LIN {X 0,Y 552.983,Z 1250.338,A -85,B 0,C 180,E1 26531.445,E2 26531.445} C_VEL
LIN {X 0,Y 553.442,Z 1236.475,A -85,B 0,C 180,E1 26529.594,E2 26529.594} C_VEL
LIN {X 0,Y 554.004,Z 1220.765,A -85,B 0,C 180,E1 26527.797,E2 26527.797} C_VEL
LIN {X 0,Y 554.663,Z 1203.891,A -85,B 0,C 180,E1 26526.129,E2 26526.129} C_VEL
LIN {X 0,Y 555.379,Z 1185.775,A -85,B 0,C 180,E1 26524.588,E2 26524.588} C_VEL
LIN {X 0,Y 556.106,Z 1167.101,A -85,B 0,C 180,E1 26523.232,E2 26523.232} C_VEL
LIN {X 0,Y 556.817,Z 1147.774,A -85,B 0,C 180,E1 26522.053,E2 26522.053} C_VEL
LIN {X 0,Y 557.493,Z 1127.887,A -85,B 0,C 180,E1 26521.038,E2 26521.038} C_VEL
LIN {X 0,Y 558.107,Z 1108.035,A -85,B 0,C 180,E1 26520.219,E2 26520.219} C_VEL
LIN {X 0,Y 558.611,Z 1086.262,A -85,B 0,C 180,E1 26519.523,E2 26519.523} C_VEL
LIN {X 0,Y 559.061,Z 1064.401,A -85,B 0,C 180,E1 26519.023,E2 26519.023} C_VEL
LIN {X 0,Y 560.686,Z 838.01,A -85,B 0,C 180,E1 26515.721,E2 26515.721} C_VEL
LIN {X 0,Y 561.006,Z 768.004,A -85,B 0,C 180,E1 26514.675,E2 26514.675} C_VEL
LIN {X 0,Y 559.471,Z 758.813,A -85,B 0,C 180,E1 26514.405,E2 26514.405} C_VEL
LIN {X 0,Y 560.826,Z 708.184,A -85,B 0,C 180,E1 26511.131,E2 26511.131} C_VEL
LIN {X 0,Y 561.473,Z 685.988,A -85,B 0,C 180,E1 26509.656,E2 26509.656} C_VEL
LIN {X 0,Y 552.413,Z 666.42,A -85,B 0,C 180,E1 26507.601,E2 26507.601} C_VEL
LIN {X 0,Y 552.326,Z 665.917,A -85,B 0,C 180,E1 26507.248,E2 26507.248} C_VEL
LIN {X 0,Y 552.322,Z 665.911,A -85,B 0,C 180,E1 26504.039,E2 26504.039} C_VEL
LIN {X 0,Y 552.331,Z 665.93,A -85,B 0,C 180,E1 26500.669,E2 26500.669} C_VEL
LIN {X 0,Y 552.333,Z 665.926,A -85,B 0,C 180,E1 26497.332,E2 26497.332} C_VEL
LIN {X 0,Y 552.336,Z 665.92,A -85,B 0,C 180,E1 26493.812,E2 26493.812} C_VEL
LIN {X 0,Y 552.328,Z 665.927,A -85,B 0,C 180,E1 26490.456,E2 26490.456} C_VEL
LIN {X 0,Y 552.327,Z 665.93,A -85,B 0,C 180,E1 26487.141,E2 26487.141} C_VEL
LIN {X 0,Y 552.324,Z 665.931,A -85,B 0,C 180,E1 26483.809,E2 26483.809} C_VEL
LIN {X 0,Y 552.324,Z 665.931,A -85,B 0,C 180,E1 26480.56,E2 26480.56} C_VEL
LIN {X 0,Y 552.323,Z 665.931,A -85,B 0,C 180,E1 26477.27,E2 26477.27} C_VEL
LIN {X 0,Y 552.324,Z 665.932,A -85,B 0,C 180,E1 26474.004,E2 26474.004} C_VEL
LIN {X 0,Y 552.324,Z 665.93,A -85,B 0,C 180,E1 26470.746,E2 26470.746} C_VEL
LIN {X 0,Y 552.327,Z 665.932,A -85,B 0,C 180,E1 26467.489,E2 26467.489} C_VEL
LIN {X 0,Y 552.325,Z 665.928,A -85,B 0,C 180,E1 26464.152,E2 26464.152} C_VEL
LIN {X 0,Y 552.345,Z 665.934,A -85,B 0,C 180,E1 26460.726,E2 26460.726} C_VEL
LIN {X 0,Y 552.337,Z 665.924,A -85,B 0,C 180,E1 26457.302,E2 26457.302} C_VEL
LIN {X 0,Y 552.332,Z 665.924,A -85,B 0,C 180,E1 26453.869,E2 26453.869} C_VEL
LIN {X 0,Y 552.335,Z 665.935,A -85,B 0,C 180,E1 26450.518,E2 26450.518} C_VEL
LIN {X 0,Y 552.324,Z 665.928,A -85,B 0,C 180,E1 26447.134,E2 26447.134} C_VEL
LIN {X 0,Y 552.341,Z 665.931,A -85,B 0,C 180,E1 26443.813,E2 26443.813} C_VEL
LIN {X 0,Y 552.326,Z 665.928,A -85,B 0,C 180,E1 26440.433,E2 26440.433} C_VEL
LIN {X 0,Y 552.338,Z 665.929,A -85,B 0,C 180,E1 26437.095,E2 26437.095} C_VEL
LIN {X 0,Y 552.336,Z 665.932,A -85,B 0,C 180,E1 26433.672,E2 26433.672} C_VEL
LIN {X 0,Y 552.339,Z 665.926,A -85,B 0,C 180,E1 26432.662,E2 26432.662} C_VEL
LIN {X 0,Y 551.37,Z 666.049,A -85,B 0,C 180,E1 26431.863,E2 26431.863} C_VEL
LIN {X 0,Y 544.853,Z 666.84,A -85,B 0,C 180,E1 26429.562,E2 26429.562} C_VEL
LIN {X 0,Y 544.401,Z 666.902,A -85,B 0,C 180,E1 26429.035,E2 26429.035} C_VEL
LIN {X 0,Y 544.387,Z 666.919,A -85,B 0,C 180,E1 26425.677,E2 26425.677} C_VEL
LIN {X 0,Y 544.387,Z 666.91,A -85,B 0,C 180,E1 26422.294,E2 26422.294} C_VEL
LIN {X 0,Y 544.386,Z 666.922,A -85,B 0,C 180,E1 26419.012,E2 26419.012} C_VEL
LIN {X 0,Y 544.387,Z 666.922,A -85,B 0,C 180,E1 26415.738,E2 26415.738} C_VEL
LIN {X 0,Y 544.393,Z 666.905,A -85,B 0,C 180,E1 26412.379,E2 26412.379} C_VEL
LIN {X 0,Y 544.391,Z 666.91,A -85,B 0,C 180,E1 26409.022,E2 26409.022} C_VEL
LIN {X 0,Y 544.427,Z 667.108,A -85,B 0,C 180,E1 26405.862,E2 26405.862} C_VEL
LIN {X 0,Y 544.787,Z 668.547,A -85,B 0,C 180,E1 26405.695,E2 26405.695} C_VEL
LIN {X 0,Y 554.114,Z 684.335,A -85,B 0,C 180,E1 26404.755,E2 26404.755} C_VEL
LIN {X 0,Y 552.272,Z 907.322,A -85,B 0,C 180,E1 26401.482,E2 26401.482} C_VEL
LIN {X 0,Y 551.925,Z 928.962,A -85,B 0,C 180,E1 26401.05,E2 26401.05} C_VEL
LIN {X 0,Y 551.302,Z 950.414,A -85,B 0,C 180,E1 26400.423,E2 26400.423} C_VEL
LIN {X 0,Y 550.639,Z 971.812,A -85,B 0,C 180,E1 26399.596,E2 26399.596} C_VEL
LIN {X 0,Y 549.869,Z 991.939,A -85,B 0,C 180,E1 26398.628,E2 26398.628} C_VEL
LIN {X 0,Y 549.069,Z 1011.113,A -85,B 0,C 180,E1 26397.497,E2 26397.497} C_VEL
LIN {X 0,Y 548.16,Z 1031.38,A -85,B 0,C 180,E1 26396.077,E2 26396.077} C_VEL
LIN {X 0,Y 547.353,Z 1049.163,A -85,B 0,C 180,E1 26394.612,E2 26394.612} C_VEL
LIN {X 0,Y 546.577,Z 1066.575,A -85,B 0,C 180,E1 26392.932,E2 26392.932} C_VEL
LIN {X 0,Y 545.879,Z 1082.44,A -85,B 0,C 180,E1 26391.151,E2 26391.151} C_VEL
LIN {X 0,Y 545.271,Z 1097.705,A -85,B 0,C 180,E1 26389.161,E2 26389.161} C_VEL
LIN {X 0,Y 544.81,Z 1110.729,A -85,B 0,C 180,E1 26387.185,E2 26387.185} C_VEL
LIN {X 0,Y 544.454,Z 1122.312,A -85,B 0,C 180,E1 26385.116,E2 26385.116} C_VEL
LIN {X 0,Y 544.213,Z 1132.49,A -85,B 0,C 180,E1 26382.952,E2 26382.952} C_VEL
LIN {X 0,Y 544.065,Z 1140.901,A -85,B 0,C 180,E1 26380.804,E2 26380.804} C_VEL
LIN {X 0,Y 543.977,Z 1147.547,A -85,B 0,C 180,E1 26378.668,E2 26378.668} C_VEL
LIN {X 0,Y 543.925,Z 1153.108,A -85,B 0,C 180,E1 26376.332,E2 26376.332} C_VEL
LIN {X 0,Y 543.908,Z 1156.822,A -85,B 0,C 180,E1 26374.111,E2 26374.111} C_VEL
LIN {X 0,Y 543.901,Z 1158.854,A -85,B 0,C 180,E1 26371.896,E2 26371.896} C_VEL
LIN {X 0,Y 543.898,Z 1159.427,A -85,B 0,C 180,E1 26369.579,E2 26369.579} C_VEL
LIN {X 0,Y 543.898,Z 1158.439,A -85,B 0,C 180,E1 26367.366,E2 26367.366} C_VEL
LIN {X 0,Y 543.904,Z 1155.79,A -85,B 0,C 180,E1 26365.11,E2 26365.11} C_VEL
LIN {X 0,Y 543.929,Z 1151.778,A -85,B 0,C 180,E1 26362.926,E2 26362.926} C_VEL
LIN {X 0,Y 543.988,Z 1146.167,A -85,B 0,C 180,E1 26360.757,E2 26360.757} C_VEL
LIN {X 0,Y 544.096,Z 1138.463,A -85,B 0,C 180,E1 26358.446,E2 26358.446} C_VEL
LIN {X 0,Y 544.28,Z 1129.612,A -85,B 0,C 180,E1 26356.292,E2 26356.292} C_VEL
LIN {X 0,Y 544.552,Z 1119.051,A -85,B 0,C 180,E1 26354.18,E2 26354.18} C_VEL
LIN {X 0,Y 544.961,Z 1106.455,A -85,B 0,C 180,E1 26352.048,E2 26352.048} C_VEL
LIN {X 0,Y 545.461,Z 1092.757,A -85,B 0,C 180,E1 26350.066,E2 26350.066} C_VEL
LIN {X 0,Y 546.099,Z 1077.486,A -85,B 0,C 180,E1 26348.167,E2 26348.167} C_VEL
LIN {X 0,Y 546.814,Z 1060.807,A -85,B 0,C 180,E1 26346.395,E2 26346.395} C_VEL
LIN {X 0,Y 547.631,Z 1042.986,A -85,B 0,C 180,E1 26344.766,E2 26344.766} C_VEL
LIN {X 0,Y 548.53,Z 1023.392,A -85,B 0,C 180,E1 26343.242,E2 26343.242} C_VEL
LIN {X 0,Y 549.377,Z 1004.059,A -85,B 0,C 180,E1 26341.969,E2 26341.969} C_VEL
LIN {X 0,Y 550.159,Z 984.662,A -85,B 0,C 180,E1 26340.913,E2 26340.913} C_VEL
LIN {X 0,Y 550.925,Z 962.845,A -85,B 0,C 180,E1 26339.941,E2 26339.941} C_VEL
LIN {X 0,Y 551.604,Z 941.595,A -85,B 0,C 180,E1 26339.203,E2 26339.203} C_VEL
LIN {X 0,Y 552.071,Z 920.027,A -85,B 0,C 180,E1 26338.66,E2 26338.66} C_VEL
LIN {X 0,Y 552.445,Z 890.261,A -85,B 0,C 180,E1 26338.174,E2 26338.174} C_VEL
LIN {X 0,Y 554.083,Z 683.904,A -85,B 0,C 180,E1 26335.146,E2 26335.146} C_VEL
LIN {X 0,Y 545.839,Z 670.561,A -85,B 0,C 180,E1 26334.331,E2 26334.331} C_VEL
LIN {X 0,Y 544.5,Z 667.51,A -85,B 0,C 180,E1 26334.127,E2 26334.127} C_VEL
LIN {X 0,Y 544.399,Z 666.917,A -85,B 0,C 180,E1 26333.876,E2 26333.876} C_VEL
LIN {X 0,Y 544.386,Z 666.914,A -85,B 0,C 180,E1 26330.48,E2 26330.48} C_VEL
LIN {X 0,Y 544.396,Z 666.906,A -85,B 0,C 180,E1 26327.123,E2 26327.123} C_VEL
LIN {X 0,Y 544.4,Z 666.909,A -85,B 0,C 180,E1 26323.676,E2 26323.676} C_VEL
LIN {X 0,Y 544.393,Z 666.919,A -85,B 0,C 180,E1 26320.18,E2 26320.18} C_VEL
LIN {X 0,Y 544.385,Z 666.904,A -85,B 0,C 180,E1 26316.781,E2 26316.781} C_VEL
LIN {X 0,Y 544.389,Z 666.922,A -85,B 0,C 180,E1 26313.436,E2 26313.436} C_VEL
LIN {X 0,Y 544.383,Z 666.898,A -85,B 0,C 180,E1 26310.094,E2 26310.094} C_VEL
LIN {X 0,Y 544.398,Z 666.922,A -85,B 0,C 180,E1 26306.742,E2 26306.742} C_VEL
LIN {X 0,Y 544.401,Z 666.915,A -85,B 0,C 180,E1 26303.258,E2 26303.258} C_VEL
LIN {X 0,Y 544.395,Z 666.919,A -85,B 0,C 180,E1 26299.752,E2 26299.752} C_VEL
LIN {X 0,Y 544.4,Z 666.919,A -85,B 0,C 180,E1 26296.43,E2 26296.43} C_VEL
LIN {X 0,Y 544.386,Z 666.918,A -85,B 0,C 180,E1 26293.057,E2 26293.057} C_VEL
LIN {X 0,Y 544.403,Z 666.922,A -85,B 0,C 180,E1 26289.728,E2 26289.728} C_VEL
LIN {X 0,Y 544.385,Z 666.912,A -85,B 0,C 180,E1 26286.433,E2 26286.433} C_VEL
LIN {X 0,Y 544.393,Z 666.918,A -85,B 0,C 180,E1 26283.053,E2 26283.053} C_VEL
LIN {X 0,Y 544.393,Z 666.919,A -85,B 0,C 180,E1 26279.684,E2 26279.684} C_VEL
LIN {X 0,Y 544.4,Z 666.917,A -85,B 0,C 180,E1 26276.209,E2 26276.209} C_VEL
LIN {X 0,Y 544.406,Z 666.918,A -85,B 0,C 180,E1 26272.72,E2 26272.72} C_VEL
LIN {X 0,Y 544.386,Z 666.918,A -85,B 0,C 180,E1 26269.292,E2 26269.292} C_VEL
LIN {X 0,Y 544.385,Z 666.919,A -85,B 0,C 180,E1 26265.97,E2 26265.97} C_VEL
LIN {X 0,Y 544.385,Z 666.92,A -85,B 0,C 180,E1 26262.69,E2 26262.69} C_VEL
LIN {X 0,Y 544.388,Z 666.919,A -85,B 0,C 180,E1 26259.351,E2 26259.351} C_VEL
LIN {X 0,Y 544.39,Z 666.918,A -85,B 0,C 180,E1 26256.053,E2 26256.053} C_VEL
LIN {X 0,Y 544.397,Z 666.918,A -85,B 0,C 180,E1 26252.667,E2 26252.667} C_VEL
LIN {X 0,Y 544.401,Z 666.922,A -85,B 0,C 180,E1 26249.175,E2 26249.175} C_VEL
LIN {X 0,Y 544.388,Z 666.911,A -85,B 0,C 180,E1 26245.738,E2 26245.738} C_VEL
LIN {X 0,Y 544.386,Z 666.914,A -85,B 0,C 180,E1 26242.427,E2 26242.427} C_VEL
LIN {X 0,Y 544.386,Z 666.911,A -85,B 0,C 180,E1 26239.167,E2 26239.167} C_VEL
LIN {X 0,Y 544.382,Z 666.897,A -85,B 0,C 180,E1 26235.885,E2 26235.885} C_VEL
LIN {X 0,Y 544.429,Z 667.133,A -85,B 0,C 180,E1 26233.02,E2 26233.02} C_VEL
LIN {X 0,Y 545.459,Z 670.023,A -85,B 0,C 180,E1 26232.688,E2 26232.688} C_VEL
LIN {X 0,Y 554.761,Z 689.588,A -85,B 0,C 180,E1 26230.644,E2 26230.644} C_VEL
LIN {X 0,Y 553.444,Z 733.168,A -85,B 0,C 180,E1 26227.765,E2 26227.765} C_VEL
LIN {X 0,Y 552.785,Z 759.73,A -85,B 0,C 180,E1 26226.062,E2 26226.062} C_VEL
LIN {X 0,Y 554.646,Z 771.849,A -85,B 0,C 180,E1 26225.732,E2 26225.732} C_VEL
LIN {X 0,Y 552.714,Z 1006.467,A -85,B 0,C 180,E1 26222.271,E2 26222.271} C_VEL
LIN {X 0,Y 552.174,Z 1066.601,A -85,B 0,C 180,E1 26221.367,E2 26221.367} C_VEL
LIN {X 0,Y 551.644,Z 1088.329,A -85,B 0,C 180,E1 26220.844,E2 26220.844} C_VEL
LIN {X 0,Y 551.02,Z 1110.245,A -85,B 0,C 180,E1 26220.113,E2 26220.113} C_VEL
LIN {X 0,Y 550.332,Z 1130.407,A -85,B 0,C 180,E1 26219.256,E2 26219.256} C_VEL
LIN {X 0,Y 549.543,Z 1149.769,A -85,B 0,C 180,E1 26218.232,E2 26218.232} C_VEL
LIN {X 0,Y 548.656,Z 1170.339,A -85,B 0,C 180,E1 26216.926,E2 26216.926} C_VEL
LIN {X 0,Y 547.804,Z 1189.118,A -85,B 0,C 180,E1 26215.514,E2 26215.514} C_VEL
LIN {X 0,Y 547.005,Z 1206.911,A -85,B 0,C 180,E1 26213.94,E2 26213.94} C_VEL
LIN {X 0,Y 546.265,Z 1223.185,A -85,B 0,C 180,E1 26212.264,E2 26212.264} C_VEL
LIN {X 0,Y 545.603,Z 1239.026,A -85,B 0,C 180,E1 26210.376,E2 26210.376} C_VEL
LIN {X 0,Y 545.098,Z 1252.633,A -85,B 0,C 180,E1 26208.501,E2 26208.501} C_VEL
LIN {X 0,Y 544.663,Z 1265.466,A -85,B 0,C 180,E1 26206.421,E2 26206.421} C_VEL
LIN {X 0,Y 544.348,Z 1276.817,A -85,B 0,C 180,E1 26204.248,E2 26204.248} C_VEL
LIN {X 0,Y 544.149,Z 1286.255,A -85,B 0,C 180,E1 26202.091,E2 26202.091} C_VEL
LIN {X 0,Y 544.023,Z 1293.885,A -85,B 0,C 180,E1 26199.948,E2 26199.948} C_VEL
LIN {X 0,Y 543.958,Z 1300.146,A -85,B 0,C 180,E1 26197.711,E2 26197.711} C_VEL
LIN {X 0,Y 543.927,Z 1304.824,A -85,B 0,C 180,E1 26195.485,E2 26195.485} C_VEL
LIN {X 0,Y 543.915,Z 1307.785,A -85,B 0,C 180,E1 26193.267,E2 26193.267} C_VEL
LIN {X 0,Y 543.906,Z 1309.306,A -85,B 0,C 180,E1 26190.948,E2 26190.948} C_VEL
LIN {X 0,Y 543.906,Z 1309.238,A -85,B 0,C 180,E1 26188.736,E2 26188.736} C_VEL
LIN {X 0,Y 543.91,Z 1307.56,A -85,B 0,C 180,E1 26186.522,E2 26186.522} C_VEL
LIN {X 0,Y 543.919,Z 1304.221,A -85,B 0,C 180,E1 26184.197,E2 26184.197} C_VEL
LIN {X 0,Y 543.959,Z 1299.636,A -85,B 0,C 180,E1 26182.076,E2 26182.076} C_VEL
LIN {X 0,Y 544.032,Z 1293.177,A -85,B 0,C 180,E1 26179.838,E2 26179.838} C_VEL
LIN {X 0,Y 544.166,Z 1285.431,A -85,B 0,C 180,E1 26177.694,E2 26177.694} C_VEL
LIN {X 0,Y 544.381,Z 1275.778,A -85,B 0,C 180,E1 26175.535,E2 26175.535} C_VEL
LIN {X 0,Y 544.708,Z 1264.197,A -85,B 0,C 180,E1 26173.361,E2 26173.361} C_VEL
LIN {X 0,Y 545.125,Z 1251.877,A -85,B 0,C 180,E1 26171.389,E2 26171.389} C_VEL
LIN {X 0,Y 545.673,Z 1237.326,A -85,B 0,C 180,E1 26169.403,E2 26169.403} C_VEL
LIN {X 0,Y 546.305,Z 1222.173,A -85,B 0,C 180,E1 26167.625,E2 26167.625} C_VEL
LIN {X 0,Y 547.107,Z 1204.496,A -85,B 0,C 180,E1 26165.836,E2 26165.836} C_VEL
LIN {X 0,Y 547.915,Z 1187.042,A -85,B 0,C 180,E1 26164.317,E2 26164.317} C_VEL
LIN {X 0,Y 548.727,Z 1168.642,A -85,B 0,C 180,E1 26162.955,E2 26162.955} C_VEL
LIN {X 0,Y 549.587,Z 1148.692,A -85,B 0,C 180,E1 26161.707,E2 26161.707} C_VEL
LIN {X 0,Y 550.381,Z 1128.624,A -85,B 0,C 180,E1 26160.662,E2 26160.662} C_VEL
LIN {X 0,Y 551.079,Z 1108.773,A -85,B 0,C 180,E1 26159.83,E2 26159.83} C_VEL
LIN {X 0,Y 551.676,Z 1086.652,A -85,B 0,C 180,E1 26159.109,E2 26159.109} C_VEL
LIN {X 0,Y 552.193,Z 1064.829,A -85,B 0,C 180,E1 26158.602,E2 26158.602} C_VEL
LIN {X 0,Y 554.061,Z 840.046,A -85,B 0,C 180,E1 26155.284,E2 26155.284} C_VEL
LIN {X 0,Y 554.469,Z 769.48,A -85,B 0,C 180,E1 26154.218,E2 26154.218} C_VEL
LIN {X 0,Y 552.702,Z 759.014,A -85,B 0,C 180,E1 26153.912,E2 26153.912} C_VEL
LIN {X 0,Y 554.316,Z 706.879,A -85,B 0,C 180,E1 26150.496,E2 26150.496} C_VEL
LIN {X 0,Y 554.76,Z 689.588,A -85,B 0,C 180,E1 26149.356,E2 26149.356} C_VEL
LIN {X 0,Y 544.48,Z 667.433,A -85,B 0,C 180,E1 26147.029,E2 26147.029} C_VEL
LIN {X 0,Y 544.389,Z 666.906,A -85,B 0,C 180,E1 26146.616,E2 26146.616} C_VEL
LIN {X 0,Y 544.388,Z 666.881,A -85,B 0,C 180,E1 26143.241,E2 26143.241} C_VEL
LIN {X 0,Y 544.386,Z 666.92,A -85,B 0,C 180,E1 26139.866,E2 26139.866} C_VEL
LIN {X 0,Y 544.388,Z 666.924,A -85,B 0,C 180,E1 26136.518,E2 26136.518} C_VEL
LIN {X 0,Y 544.389,Z 666.913,A -85,B 0,C 180,E1 26133.183,E2 26133.183} C_VEL
LIN {X 0,Y 544.399,Z 666.906,A -85,B 0,C 180,E1 26129.728,E2 26129.728} C_VEL
LIN {X 0,Y 544.395,Z 666.92,A -85,B 0,C 180,E1 26126.272,E2 26126.272} C_VEL
LIN {X 0,Y 544.392,Z 666.916,A -85,B 0,C 180,E1 26122.915,E2 26122.915} C_VEL
LIN {X 0,Y 544.386,Z 666.909,A -85,B 0,C 180,E1 26119.528,E2 26119.528} C_VEL
LIN {X 0,Y 544.385,Z 666.922,A -85,B 0,C 180,E1 26116.211,E2 26116.211} C_VEL
LIN {X 0,Y 544.384,Z 666.908,A -85,B 0,C 180,E1 26112.948,E2 26112.948} C_VEL
LIN {X 0,Y 544.388,Z 666.925,A -85,B 0,C 180,E1 26109.621,E2 26109.621} C_VEL
LIN {X 0,Y 544.386,Z 666.917,A -85,B 0,C 180,E1 26106.327,E2 26106.327} C_VEL
LIN {X 0,Y 544.403,Z 666.918,A -85,B 0,C 180,E1 26102.948,E2 26102.948} C_VEL
LIN {X 0,Y 544.404,Z 666.917,A -85,B 0,C 180,E1 26099.474,E2 26099.474} C_VEL
LIN {X 0,Y 544.393,Z 666.919,A -85,B 0,C 180,E1 26095.998,E2 26095.998} C_VEL
LIN {X 0,Y 544.392,Z 666.917,A -85,B 0,C 180,E1 26092.64,E2 26092.64} C_VEL
LIN {X 0,Y 544.386,Z 666.914,A -85,B 0,C 180,E1 26089.293,E2 26089.293} C_VEL
LIN {X 0,Y 544.404,Z 666.923,A -85,B 0,C 180,E1 26085.97,E2 26085.97} C_VEL
LIN {X 0,Y 544.388,Z 666.917,A -85,B 0,C 180,E1 26082.58,E2 26082.58} C_VEL
LIN {X 0,Y 544.402,Z 666.916,A -85,B 0,C 180,E1 26079.126,E2 26079.126} C_VEL
LIN {X 0,Y 544.402,Z 666.919,A -85,B 0,C 180,E1 26075.707,E2 26075.707} C_VEL
LIN {X 0,Y 544.391,Z 666.915,A -85,B 0,C 180,E1 26072.281,E2 26072.281} C_VEL
LIN {X 0,Y 544.401,Z 666.902,A -85,B 0,C 180,E1 26069.035,E2 26069.035} C_VEL
LIN {X 0,Y 543.391,Z 667.039,A -85,B 0,C 180,E1 26068.224,E2 26068.224} C_VEL
LIN {X 0,Y 536.973,Z 667.844,A -85,B 0,C 180,E1 26065.948,E2 26065.948} C_VEL
LIN {X 0,Y 536.45,Z 667.911,A -85,B 0,C 180,E1 26065.354,E2 26065.354} C_VEL
LIN {X 0,Y 536.461,Z 667.9,A -85,B 0,C 180,E1 26061.86,E2 26061.86} C_VEL
LIN {X 0,Y 536.456,Z 667.895,A -85,B 0,C 180,E1 26058.363,E2 26058.363} C_VEL
LIN {X 0,Y 536.452,Z 667.911,A -85,B 0,C 180,E1 26054.907,E2 26054.907} C_VEL
LIN {X 0,Y 536.447,Z 667.899,A -85,B 0,C 180,E1 26051.568,E2 26051.568} C_VEL
LIN {X 0,Y 536.454,Z 667.894,A -85,B 0,C 180,E1 26048.227,E2 26048.227} C_VEL
LIN {X 0,Y 536.505,Z 668.21,A -85,B 0,C 180,E1 26046.44,E2 26046.44} C_VEL
LIN {X 0,Y 536.67,Z 668.989,A -85,B 0,C 180,E1 26046.33,E2 26046.33} C_VEL
LIN {X 0,Y 538.429,Z 672.229,A -85,B 0,C 180,E1 26046.119,E2 26046.119} C_VEL
LIN {X 0,Y 547.517,Z 687.437,A -85,B 0,C 180,E1 26045.187,E2 26045.187} C_VEL
LIN {X 0,Y 545.382,Z 912.875,A -85,B 0,C 180,E1 26041.827,E2 26041.827} C_VEL
LIN {X 0,Y 544.835,Z 935.388,A -85,B 0,C 180,E1 26041.314,E2 26041.314} C_VEL
LIN {X 0,Y 544.207,Z 956.203,A -85,B 0,C 180,E1 26040.652,E2 26040.652} C_VEL
LIN {X 0,Y 543.439,Z 975.676,A -85,B 0,C 180,E1 26039.846,E2 26039.846} C_VEL
LIN {X 0,Y 542.495,Z 997.018,A -85,B 0,C 180,E1 26038.752,E2 26038.752} C_VEL
LIN {X 0,Y 541.569,Z 1016.484,A -85,B 0,C 180,E1 26037.546,E2 26037.546} C_VEL
LIN {X 0,Y 540.615,Z 1035.042,A -85,B 0,C 180,E1 26036.173,E2 26036.173} C_VEL
LIN {X 0,Y 539.637,Z 1053.486,A -85,B 0,C 180,E1 26034.573,E2 26034.573} C_VEL
LIN {X 0,Y 538.756,Z 1070.763,A -85,B 0,C 180,E1 26032.822,E2 26032.822} C_VEL
LIN {X 0,Y 538.031,Z 1086.136,A -85,B 0,C 180,E1 26031.018,E2 26031.018} C_VEL
LIN {X 0,Y 537.359,Z 1100.798,A -85,B 0,C 180,E1 26029.003,E2 26029.003} C_VEL
LIN {X 0,Y 536.859,Z 1113.299,A -85,B 0,C 180,E1 26027.001,E2 26027.001} C_VEL
LIN {X 0,Y 536.48,Z 1124.531,A -85,B 0,C 180,E1 26024.903,E2 26024.903} C_VEL
LIN {X 0,Y 536.228,Z 1134.005,A -85,B 0,C 180,E1 26022.788,E2 26022.788} C_VEL
LIN {X 0,Y 536.059,Z 1142.323,A -85,B 0,C 180,E1 26020.532,E2 26020.532} C_VEL
LIN {X 0,Y 535.967,Z 1149.023,A -85,B 0,C 180,E1 26018.259,E2 26018.259} C_VEL
LIN {X 0,Y 535.918,Z 1153.932,A -85,B 0,C 180,E1 26015.997,E2 26015.997} C_VEL
LIN {X 0,Y 535.901,Z 1157.402,A -85,B 0,C 180,E1 26013.637,E2 26013.637} C_VEL
LIN {X 0,Y 535.899,Z 1159.188,A -85,B 0,C 180,E1 26011.39,E2 26011.39} C_VEL
LIN {X 0,Y 535.902,Z 1159.338,A -85,B 0,C 180,E1 26009.145,E2 26009.145} C_VEL
LIN {X 0,Y 535.912,Z 1157.946,A -85,B 0,C 180,E1 26006.791,E2 26006.791} C_VEL
LIN {X 0,Y 535.923,Z 1155.052,A -85,B 0,C 180,E1 26004.54,E2 26004.54} C_VEL
LIN {X 0,Y 535.953,Z 1150.506,A -85,B 0,C 180,E1 26002.281,E2 26002.281} C_VEL
LIN {X 0,Y 536.031,Z 1144.384,A -85,B 0,C 180,E1 26000.011,E2 26000.011} C_VEL
LIN {X 0,Y 536.171,Z 1136.83,A -85,B 0,C 180,E1 25997.836,E2 25997.836} C_VEL
LIN {X 0,Y 536.42,Z 1127.03,A -85,B 0,C 180,E1 25995.537,E2 25995.537} C_VEL
LIN {X 0,Y 536.783,Z 1115.722,A -85,B 0,C 180,E1 25993.331,E2 25993.331} C_VEL
LIN {X 0,Y 537.249,Z 1103.512,A -85,B 0,C 180,E1 25991.314,E2 25991.314} C_VEL
LIN {X 0,Y 537.853,Z 1089.36,A -85,B 0,C 180,E1 25989.317,E2 25989.317} C_VEL
LIN {X 0,Y 538.609,Z 1073.587,A -85,B 0,C 180,E1 25987.402,E2 25987.402} C_VEL
LIN {X 0,Y 539.481,Z 1056.976,A -85,B 0,C 180,E1 25985.665,E2 25985.665} C_VEL
LIN {X 0,Y 540.372,Z 1039.626,A -85,B 0,C 180,E1 25984.109,E2 25984.109} C_VEL
LIN {X 0,Y 541.328,Z 1020.931,A -85,B 0,C 180,E1 25982.677,E2 25982.677} C_VEL
LIN {X 0,Y 542.351,Z 1000.312,A -85,B 0,C 180,E1 25981.347,E2 25981.347} C_VEL
LIN {X 0,Y 543.259,Z 980.1,A -85,B 0,C 180,E1 25980.265,E2 25980.265} C_VEL
LIN {X 0,Y 544.064,Z 959.86,A -85,B 0,C 180,E1 25979.4,E2 25979.4} C_VEL
LIN {X 0,Y 544.758,Z 937.923,A -85,B 0,C 180,E1 25978.665,E2 25978.665} C_VEL
LIN {X 0,Y 545.35,Z 916.042,A -85,B 0,C 180,E1 25978.139,E2 25978.139} C_VEL
LIN {X 0,Y 546.247,Z 823.488,A -85,B 0,C 180,E1 25976.749,E2 25976.749} C_VEL
LIN {X 0,Y 547.417,Z 686.99,A -85,B 0,C 180,E1 25974.708,E2 25974.708} C_VEL
LIN {X 0,Y 538.242,Z 672.015,A -85,B 0,C 180,E1 25973.773,E2 25973.773} C_VEL
LIN {X 0,Y 536.623,Z 668.787,A -85,B 0,C 180,E1 25973.56,E2 25973.56} C_VEL
LIN {X 0,Y 536.479,Z 668.01,A -85,B 0,C 180,E1 25973.389,E2 25973.389} C_VEL
LIN {X 0,Y 536.463,Z 667.908,A -85,B 0,C 180,E1 25969.985,E2 25969.985} C_VEL
LIN {X 0,Y 536.449,Z 667.899,A -85,B 0,C 180,E1 25966.549,E2 25966.549} C_VEL
LIN {X 0,Y 536.45,Z 667.887,A -85,B 0,C 180,E1 25963.16,E2 25963.16} C_VEL
LIN {X 0,Y 536.448,Z 667.911,A -85,B 0,C 180,E1 25959.836,E2 25959.836} C_VEL
LIN {X 0,Y 536.447,Z 667.891,A -85,B 0,C 180,E1 25956.482,E2 25956.482} C_VEL
LIN {X 0,Y 536.46,Z 667.915,A -85,B 0,C 180,E1 25953.1,E2 25953.1} C_VEL
LIN {X 0,Y 536.463,Z 667.882,A -85,B 0,C 180,E1 25949.598,E2 25949.598} C_VEL
LIN {X 0,Y 536.455,Z 667.91,A -85,B 0,C 180,E1 25946.214,E2 25946.214} C_VEL
LIN {X 0,Y 536.457,Z 667.907,A -85,B 0,C 180,E1 25942.81,E2 25942.81} C_VEL
LIN {X 0,Y 536.448,Z 667.906,A -85,B 0,C 180,E1 25939.425,E2 25939.425} C_VEL
LIN {X 0,Y 536.462,Z 667.906,A -85,B 0,C 180,E1 25936.012,E2 25936.012} C_VEL
LIN {X 0,Y 536.455,Z 667.906,A -85,B 0,C 180,E1 25932.596,E2 25932.596} C_VEL
LIN {X 0,Y 536.463,Z 667.908,A -85,B 0,C 180,E1 25929.116,E2 25929.116} C_VEL
LIN {X 0,Y 536.465,Z 667.904,A -85,B 0,C 180,E1 25925.669,E2 25925.669} C_VEL
LIN {X 0,Y 536.447,Z 667.9,A -85,B 0,C 180,E1 25922.243,E2 25922.243} C_VEL
LIN {X 0,Y 536.455,Z 667.912,A -85,B 0,C 180,E1 25918.932,E2 25918.932} C_VEL
LIN {X 0,Y 536.446,Z 667.907,A -85,B 0,C 180,E1 25915.617,E2 25915.617} C_VEL
LIN {X 0,Y 536.449,Z 667.908,A -85,B 0,C 180,E1 25912.288,E2 25912.288} C_VEL
LIN {X 0,Y 536.454,Z 667.909,A -85,B 0,C 180,E1 25908.932,E2 25908.932} C_VEL
LIN {X 0,Y 536.463,Z 667.902,A -85,B 0,C 180,E1 25905.427,E2 25905.427} C_VEL
LIN {X 0,Y 536.455,Z 667.901,A -85,B 0,C 180,E1 25901.977,E2 25901.977} C_VEL
LIN {X 0,Y 536.448,Z 667.908,A -85,B 0,C 180,E1 25898.573,E2 25898.573} C_VEL
LIN {X 0,Y 536.446,Z 667.901,A -85,B 0,C 180,E1 25895.206,E2 25895.206} C_VEL
LIN {X 0,Y 536.448,Z 667.913,A -85,B 0,C 180,E1 25891.833,E2 25891.833} C_VEL
LIN {X 0,Y 536.456,Z 667.908,A -85,B 0,C 180,E1 25888.401,E2 25888.401} C_VEL
LIN {X 0,Y 536.461,Z 667.91,A -85,B 0,C 180,E1 25884.903,E2 25884.903} C_VEL
LIN {X 0,Y 536.455,Z 667.904,A -85,B 0,C 180,E1 25881.5,E2 25881.5} C_VEL
LIN {X 0,Y 536.445,Z 667.874,A -85,B 0,C 180,E1 25878.144,E2 25878.144} C_VEL
LIN {X 0,Y 536.451,Z 667.914,A -85,B 0,C 180,E1 25874.79,E2 25874.79} C_VEL
LIN {X 0,Y 536.481,Z 668.149,A -85,B 0,C 180,E1 25873.616,E2 25873.616} C_VEL
LIN {X 0,Y 537.828,Z 671.478,A -85,B 0,C 180,E1 25873.218,E2 25873.218} C_VEL
LIN {X 0,Y 547.876,Z 693.104,A -85,B 0,C 180,E1 25870.928,E2 25870.928} C_VEL
LIN {X 0,Y 546.966,Z 729.324,A -85,B 0,C 180,E1 25868.56,E2 25868.56} C_VEL
LIN {X 0,Y 546.041,Z 759.689,A -85,B 0,C 180,E1 25866.579,E2 25866.579} C_VEL
LIN {X 0,Y 548.138,Z 773.248,A -85,B 0,C 180,E1 25866.201,E2 25866.201} C_VEL
LIN {X 0,Y 545.942,Z 1007.485,A -85,B 0,C 180,E1 25862.705,E2 25862.705} C_VEL
LIN {X 0,Y 545.334,Z 1066.781,A -85,B 0,C 180,E1 25861.803,E2 25861.803} C_VEL
LIN {X 0,Y 544.737,Z 1088.59,A -85,B 0,C 180,E1 25861.271,E2 25861.271} C_VEL
LIN {X 0,Y 544.044,Z 1110.242,A -85,B 0,C 180,E1 25860.54,E2 25860.54} C_VEL
LIN {X 0,Y 543.255,Z 1130.406,A -85,B 0,C 180,E1 25859.675,E2 25859.675} C_VEL
LIN {X 0,Y 542.369,Z 1149.772,A -85,B 0,C 180,E1 25858.639,E2 25858.639} C_VEL
LIN {X 0,Y 541.361,Z 1170.18,A -85,B 0,C 180,E1 25857.331,E2 25857.331} C_VEL
LIN {X 0,Y 540.405,Z 1189.115,A -85,B 0,C 180,E1 25855.889,E2 25855.889} C_VEL
LIN {X 0,Y 539.481,Z 1206.913,A -85,B 0,C 180,E1 25854.295,E2 25854.295} C_VEL
LIN {X 0,Y 538.628,Z 1223.185,A -85,B 0,C 180,E1 25852.597,E2 25852.597} C_VEL
LIN {X 0,Y 537.869,Z 1239.027,A -85,B 0,C 180,E1 25850.682,E2 25850.682} C_VEL
LIN {X 0,Y 537.265,Z 1253.19,A -85,B 0,C 180,E1 25848.692,E2 25848.692} C_VEL
LIN {X 0,Y 536.793,Z 1265.464,A -85,B 0,C 180,E1 25846.669,E2 25846.669} C_VEL
LIN {X 0,Y 536.428,Z 1276.818,A -85,B 0,C 180,E1 25844.463,E2 25844.463} C_VEL
LIN {X 0,Y 536.187,Z 1286.256,A -85,B 0,C 180,E1 25842.273,E2 25842.273} C_VEL
LIN {X 0,Y 536.042,Z 1293.884,A -85,B 0,C 180,E1 25840.098,E2 25840.098} C_VEL
LIN {X 0,Y 535.964,Z 1300.146,A -85,B 0,C 180,E1 25837.827,E2 25837.827} C_VEL
LIN {X 0,Y 535.928,Z 1304.824,A -85,B 0,C 180,E1 25835.567,E2 25835.567} C_VEL
LIN {X 0,Y 535.915,Z 1307.786,A -85,B 0,C 180,E1 25833.316,E2 25833.316} C_VEL
LIN {X 0,Y 535.907,Z 1309.306,A -85,B 0,C 180,E1 25830.962,E2 25830.962} C_VEL
LIN {X 0,Y 535.905,Z 1309.237,A -85,B 0,C 180,E1 25828.717,E2 25828.717} C_VEL
LIN {X 0,Y 535.906,Z 1307.56,A -85,B 0,C 180,E1 25826.47,E2 25826.47} C_VEL
LIN {X 0,Y 535.922,Z 1304.427,A -85,B 0,C 180,E1 25824.218,E2 25824.218} C_VEL
LIN {X 0,Y 535.963,Z 1299.891,A -85,B 0,C 180,E1 25822.065,E2 25822.065} C_VEL
LIN {X 0,Y 536.047,Z 1293.177,A -85,B 0,C 180,E1 25819.685,E2 25819.685} C_VEL
LIN {X 0,Y 536.203,Z 1285.431,A -85,B 0,C 180,E1 25817.508,E2 25817.508} C_VEL
LIN {X 0,Y 536.45,Z 1275.765,A -85,B 0,C 180,E1 25815.314,E2 25815.314} C_VEL
LIN {X 0,Y 536.836,Z 1264.195,A -85,B 0,C 180,E1 25813.11,E2 25813.11} C_VEL
LIN {X 0,Y 537.323,Z 1251.875,A -85,B 0,C 180,E1 25811.109,E2 25811.109} C_VEL
LIN {X 0,Y 537.958,Z 1237.327,A -85,B 0,C 180,E1 25809.094,E2 25809.094} C_VEL
LIN {X 0,Y 538.676,Z 1222.172,A -85,B 0,C 180,E1 25807.29,E2 25807.29} C_VEL
LIN {X 0,Y 539.593,Z 1204.498,A -85,B 0,C 180,E1 25805.477,E2 25805.477} C_VEL
LIN {X 0,Y 540.509,Z 1187.311,A -85,B 0,C 180,E1 25803.961,E2 25803.961} C_VEL
LIN {X 0,Y 541.434,Z 1168.716,A -85,B 0,C 180,E1 25802.566,E2 25802.566} C_VEL
LIN {X 0,Y 542.408,Z 1148.874,A -85,B 0,C 180,E1 25801.309,E2 25801.309} C_VEL
LIN {X 0,Y 543.3,Z 1129.168,A -85,B 0,C 180,E1 25800.267,E2 25800.267} C_VEL
LIN {X 0,Y 544.076,Z 1109.51,A -85,B 0,C 180,E1 25799.431,E2 25799.431} C_VEL
LIN {X 0,Y 544.773,Z 1087.041,A -85,B 0,C 180,E1 25798.685,E2 25798.685} C_VEL
LIN {X 0,Y 545.354,Z 1065.365,A -85,B 0,C 180,E1 25798.172,E2 25798.172} C_VEL
LIN {X 0,Y 547.157,Z 872.798,A -85,B 0,C 180,E1 25795.296,E2 25795.296} C_VEL
LIN {X 0,Y 547.969,Z 770.942,A -85,B 0,C 180,E1 25793.749,E2 25793.749} C_VEL
LIN {X 0,Y 545.964,Z 758.712,A -85,B 0,C 180,E1 25793.377,E2 25793.377} C_VEL
LIN {X 0,Y 547.518,Z 711.153,A -85,B 0,C 180,E1 25790.247,E2 25790.247} C_VEL
LIN {X 0,Y 547.847,Z 693.046,A -85,B 0,C 180,E1 25789.067,E2 25789.067} C_VEL
LIN {X 0,Y 536.528,Z 668.422,A -85,B 0,C 180,E1 25786.432,E2 25786.432} C_VEL
LIN {X 0,Y 536.457,Z 667.902,A -85,B 0,C 180,E1 25785.958,E2 25785.958} C_VEL
LIN {X 0,Y 536.454,Z 667.865,A -85,B 0,C 180,E1 25782.431,E2 25782.431} C_VEL
LIN {X 0,Y 536.456,Z 667.91,A -85,B 0,C 180,E1 25778.996,E2 25778.996} C_VEL
LIN {X 0,Y 536.446,Z 667.911,A -85,B 0,C 180,E1 25775.648,E2 25775.648} C_VEL
LIN {X 0,Y 536.449,Z 667.913,A -85,B 0,C 180,E1 25772.338,E2 25772.338} C_VEL
LIN {X 0,Y 536.448,Z 667.898,A -85,B 0,C 180,E1 25768.986,E2 25768.986} C_VEL
LIN {X 0,Y 536.454,Z 667.9,A -85,B 0,C 180,E1 25765.569,E2 25765.569} C_VEL
LIN {X 0,Y 536.466,Z 667.914,A -85,B 0,C 180,E1 25762.116,E2 25762.116} C_VEL
LIN {X 0,Y 536.454,Z 667.893,A -85,B 0,C 180,E1 25758.698,E2 25758.698} C_VEL
LIN {X 0,Y 536.452,Z 667.907,A -85,B 0,C 180,E1 25755.347,E2 25755.347} C_VEL
LIN {X 0,Y 536.448,Z 667.897,A -85,B 0,C 180,E1 25752.049,E2 25752.049} C_VEL
LIN {X 0,Y 536.446,Z 667.906,A -85,B 0,C 180,E1 25748.683,E2 25748.683} C_VEL
LIN {X 0,Y 536.451,Z 667.913,A -85,B 0,C 180,E1 25745.347,E2 25745.347} C_VEL
LIN {X 0,Y 536.451,Z 667.903,A -85,B 0,C 180,E1 25741.922,E2 25741.922} C_VEL
LIN {X 0,Y 536.467,Z 667.902,A -85,B 0,C 180,E1 25738.505,E2 25738.505} C_VEL
LIN {X 0,Y 536.459,Z 667.909,A -85,B 0,C 180,E1 25735.081,E2 25735.081} C_VEL
LIN {X 0,Y 536.452,Z 667.907,A -85,B 0,C 180,E1 25731.641,E2 25731.641} C_VEL
LIN {X 0,Y 536.459,Z 667.906,A -85,B 0,C 180,E1 25728.278,E2 25728.278} C_VEL
LIN {X 0,Y 536.447,Z 667.905,A -85,B 0,C 180,E1 25724.874,E2 25724.874} C_VEL
LIN {X 0,Y 536.463,Z 667.909,A -85,B 0,C 180,E1 25721.528,E2 25721.528} C_VEL
LIN {X 0,Y 536.456,Z 667.907,A -85,B 0,C 180,E1 25718.114,E2 25718.114} C_VEL
LIN {X 0,Y 536.461,Z 667.905,A -85,B 0,C 180,E1 25714.616,E2 25714.616} C_VEL
LIN {X 0,Y 536.463,Z 667.891,A -85,B 0,C 180,E1 25711.136,E2 25711.136} C_VEL
LIN {X 0,Y 536.447,Z 667.902,A -85,B 0,C 180,E1 25707.787,E2 25707.787} C_VEL
LIN {X 0,Y 536.45,Z 667.911,A -85,B 0,C 180,E1 25705.354,E2 25705.354} C_VEL
LIN {X 0,Y 535.479,Z 668.037,A -85,B 0,C 180,E1 25704.532,E2 25704.532} C_VEL
LIN {X 0,Y 528.975,Z 668.833,A -85,B 0,C 180,E1 25702.161,E2 25702.161} C_VEL
LIN {X 0,Y 528.519,Z 668.889,A -85,B 0,C 180,E1 25701.618,E2 25701.618} C_VEL
LIN {X 0,Y 528.51,Z 668.88,A -85,B 0,C 180,E1 25698.19,E2 25698.19} C_VEL
LIN {X 0,Y 528.512,Z 668.901,A -85,B 0,C 180,E1 25694.811,E2 25694.811} C_VEL
LIN {X 0,Y 528.507,Z 668.888,A -85,B 0,C 180,E1 25691.462,E2 25691.462} C_VEL
LIN {X 0,Y 528.519,Z 668.881,A -85,B 0,C 180,E1 25688.076,E2 25688.076} C_VEL
LIN {X 0,Y 528.552,Z 669.188,A -85,B 0,C 180,E1 25687.081,E2 25687.081} C_VEL
LIN {X 0,Y 528.971,Z 670.747,A -85,B 0,C 180,E1 25686.912,E2 25686.912} C_VEL
LIN {X 0,Y 537.01,Z 683.747,A -85,B 0,C 180,E1 25686.043,E2 25686.043} C_VEL
LIN {X 0,Y 540.95,Z 690.544,A -85,B 0,C 180,E1 25685.63,E2 25685.63} C_VEL
LIN {X 0,Y 538.571,Z 913.989,A -85,B 0,C 180,E1 25682.258,E2 25682.258} C_VEL
LIN {X 0,Y 537.964,Z 935.935,A -85,B 0,C 180,E1 25681.745,E2 25681.745} C_VEL
LIN {X 0,Y 537.239,Z 956.959,A -85,B 0,C 180,E1 25681.063,E2 25681.063} C_VEL
LIN {X 0,Y 536.367,Z 976.968,A -85,B 0,C 180,E1 25680.219,E2 25680.219} C_VEL
LIN {X 0,Y 535.36,Z 997.028,A -85,B 0,C 180,E1 25679.172,E2 25679.172} C_VEL
LIN {X 0,Y 534.351,Z 1016.231,A -85,B 0,C 180,E1 25677.97,E2 25677.97} C_VEL
LIN {X 0,Y 533.262,Z 1034.932,A -85,B 0,C 180,E1 25676.572,E2 25676.572} C_VEL
LIN {X 0,Y 532.192,Z 1052.823,A -85,B 0,C 180,E1 25675.006,E2 25675.006} C_VEL
LIN {X 0,Y 531.236,Z 1069.756,A -85,B 0,C 180,E1 25673.281,E2 25673.281} C_VEL
LIN {X 0,Y 530.378,Z 1085.225,A -85,B 0,C 180,E1 25671.452,E2 25671.452} C_VEL
LIN {X 0,Y 529.645,Z 1099.261,A -85,B 0,C 180,E1 25669.52,E2 25669.52} C_VEL
LIN {X 0,Y 529.022,Z 1112.754,A -85,B 0,C 180,E1 25667.358,E2 25667.358} C_VEL
LIN {X 0,Y 528.591,Z 1124.016,A -85,B 0,C 180,E1 25665.243,E2 25665.243} C_VEL
LIN {X 0,Y 528.283,Z 1133.876,A -85,B 0,C 180,E1 25663.016,E2 25663.016} C_VEL
LIN {X 0,Y 528.083,Z 1142.352,A -85,B 0,C 180,E1 25660.685,E2 25660.685} C_VEL
LIN {X 0,Y 527.976,Z 1149.024,A -85,B 0,C 180,E1 25658.384,E2 25658.384} C_VEL
LIN {X 0,Y 527.921,Z 1153.934,A -85,B 0,C 180,E1 25656.088,E2 25656.088} C_VEL
LIN {X 0,Y 527.9,Z 1157.402,A -85,B 0,C 180,E1 25653.692,E2 25653.692} C_VEL
LIN {X 0,Y 527.898,Z 1159.188,A -85,B 0,C 180,E1 25651.411,E2 25651.411} C_VEL
LIN {X 0,Y 527.903,Z 1159.337,A -85,B 0,C 180,E1 25649.132,E2 25649.132} C_VEL
LIN {X 0,Y 527.914,Z 1157.945,A -85,B 0,C 180,E1 25646.743,E2 25646.743} C_VEL
LIN {X 0,Y 527.927,Z 1155.051,A -85,B 0,C 180,E1 25644.457,E2 25644.457} C_VEL
LIN {X 0,Y 527.957,Z 1150.504,A -85,B 0,C 180,E1 25642.163,E2 25642.163} C_VEL
LIN {X 0,Y 528.051,Z 1144.382,A -85,B 0,C 180,E1 25639.858,E2 25639.858} C_VEL
LIN {X 0,Y 528.21,Z 1136.828,A -85,B 0,C 180,E1 25637.649,E2 25637.649} C_VEL
LIN {X 0,Y 528.495,Z 1127.026,A -85,B 0,C 180,E1 25635.315,E2 25635.315} C_VEL
LIN {X 0,Y 528.913,Z 1115.717,A -85,B 0,C 180,E1 25633.075,E2 25633.075} C_VEL
LIN {X 0,Y 529.442,Z 1103.62,A -85,B 0,C 180,E1 25631.046,E2 25631.046} C_VEL
LIN {X 0,Y 530.092,Z 1090.203,A -85,B 0,C 180,E1 25629.116,E2 25629.116} C_VEL
LIN {X 0,Y 530.94,Z 1074.594,A -85,B 0,C 180,E1 25627.175,E2 25627.175} C_VEL
LIN {X 0,Y 531.892,Z 1058.561,A -85,B 0,C 180,E1 25625.454,E2 25625.454} C_VEL
LIN {X 0,Y 532.901,Z 1040.954,A -85,B 0,C 180,E1 25623.838,E2 25623.838} C_VEL
LIN {X 0,Y 534.012,Z 1021.695,A -85,B 0,C 180,E1 25622.328,E2 25622.328} C_VEL
LIN {X 0,Y 535.099,Z 1002.503,A -85,B 0,C 180,E1 25621.057,E2 25621.057} C_VEL
LIN {X 0,Y 536.045,Z 983.491,A -85,B 0,C 180,E1 25620.008,E2 25620.008} C_VEL
LIN {X 0,Y 536.991,Z 962.804,A -85,B 0,C 180,E1 25619.077,E2 25619.077} C_VEL
LIN {X 0,Y 537.808,Z 941.925,A -85,B 0,C 180,E1 25618.335,E2 25618.335} C_VEL
LIN {X 0,Y 538.413,Z 920.286,A -85,B 0,C 180,E1 25617.779,E2 25617.779} C_VEL
LIN {X 0,Y 538.876,Z 890.668,A -85,B 0,C 180,E1 25617.282,E2 25617.282} C_VEL
LIN {X 0,Y 540.89,Z 690.014,A -85,B 0,C 180,E1 25614.267,E2 25614.267} C_VEL
LIN {X 0,Y 530.371,Z 673.11,A -85,B 0,C 180,E1 25613.165,E2 25613.165} C_VEL
LIN {X 0,Y 528.644,Z 669.671,A -85,B 0,C 180,E1 25612.918,E2 25612.918} C_VEL
LIN {X 0,Y 528.522,Z 668.994,A -85,B 0,C 180,E1 25612.745,E2 25612.745} C_VEL
LIN {X 0,Y 528.521,Z 668.9,A -85,B 0,C 180,E1 25609.342,E2 25609.342} C_VEL
LIN {X 0,Y 528.521,Z 668.893,A -85,B 0,C 180,E1 25605.88,E2 25605.88} C_VEL
LIN {X 0,Y 528.514,Z 668.87,A -85,B 0,C 180,E1 25602.337,E2 25602.337} C_VEL
LIN {X 0,Y 528.511,Z 668.895,A -85,B 0,C 180,E1 25598.91,E2 25598.91} C_VEL
LIN {X 0,Y 528.509,Z 668.884,A -85,B 0,C 180,E1 25595.507,E2 25595.507} C_VEL
LIN {X 0,Y 528.511,Z 668.89,A -85,B 0,C 180,E1 25592.114,E2 25592.114} C_VEL
LIN {X 0,Y 528.525,Z 668.882,A -85,B 0,C 180,E1 25588.596,E2 25588.596} C_VEL
LIN {X 0,Y 528.52,Z 668.896,A -85,B 0,C 180,E1 25585.073,E2 25585.073} C_VEL
LIN {X 0,Y 528.509,Z 668.895,A -85,B 0,C 180,E1 25581.649,E2 25581.649} C_VEL
LIN {X 0,Y 528.524,Z 668.902,A -85,B 0,C 180,E1 25578.189,E2 25578.189} C_VEL
LIN {X 0,Y 528.521,Z 668.893,A -85,B 0,C 180,E1 25574.685,E2 25574.685} C_VEL
LIN {X 0,Y 528.516,Z 668.893,A -85,B 0,C 180,E1 25571.126,E2 25571.126} C_VEL
LIN {X 0,Y 528.53,Z 668.896,A -85,B 0,C 180,E1 25567.61,E2 25567.61} C_VEL
LIN {X 0,Y 528.508,Z 668.897,A -85,B 0,C 180,E1 25564.231,E2 25564.231} C_VEL
LIN {X 0,Y 528.517,Z 668.9,A -85,B 0,C 180,E1 25560.759,E2 25560.759} C_VEL
LIN {X 0,Y 528.524,Z 668.893,A -85,B 0,C 180,E1 25557.289,E2 25557.289} C_VEL
LIN {X 0,Y 528.514,Z 668.894,A -85,B 0,C 180,E1 25553.81,E2 25553.81} C_VEL
LIN {X 0,Y 528.515,Z 668.904,A -85,B 0,C 180,E1 25550.417,E2 25550.417} C_VEL
LIN {X 0,Y 528.506,Z 668.883,A -85,B 0,C 180,E1 25547.101,E2 25547.101} C_VEL
LIN {X 0,Y 528.509,Z 668.9,A -85,B 0,C 180,E1 25543.74,E2 25543.74} C_VEL
LIN {X 0,Y 528.513,Z 668.884,A -85,B 0,C 180,E1 25540.321,E2 25540.321} C_VEL
LIN {X 0,Y 528.525,Z 668.892,A -85,B 0,C 180,E1 25536.828,E2 25536.828} C_VEL
LIN {X 0,Y 528.514,Z 668.904,A -85,B 0,C 180,E1 25533.362,E2 25533.362} C_VEL
LIN {X 0,Y 528.508,Z 668.885,A -85,B 0,C 180,E1 25530.037,E2 25530.037} C_VEL
LIN {X 0,Y 528.509,Z 668.888,A -85,B 0,C 180,E1 25526.727,E2 25526.727} C_VEL
LIN {X 0,Y 528.509,Z 668.9,A -85,B 0,C 180,E1 25523.333,E2 25523.333} C_VEL
LIN {X 0,Y 528.51,Z 668.898,A -85,B 0,C 180,E1 25519.967,E2 25519.967} C_VEL
LIN {X 0,Y 528.523,Z 668.85,A -85,B 0,C 180,E1 25516.48,E2 25516.48} C_VEL
LIN {X 0,Y 528.565,Z 669.161,A -85,B 0,C 180,E1 25514.234,E2 25514.234} C_VEL
LIN {X 0,Y 529.967,Z 672.612,A -85,B 0,C 180,E1 25513.81,E2 25513.81} C_VEL
LIN {X 0,Y 541.051,Z 696.868,A -85,B 0,C 180,E1 25511.198,E2 25511.198} C_VEL
LIN {X 0,Y 539.79,Z 744.841,A -85,B 0,C 180,E1 25508.073,E2 25508.073} C_VEL
LIN {X 0,Y 539.363,Z 759.811,A -85,B 0,C 180,E1 25507.106,E2 25507.106} C_VEL
LIN {X 0,Y 541.668,Z 774.71,A -85,B 0,C 180,E1 25506.68,E2 25506.68} C_VEL
LIN {X 0,Y 539.204,Z 1008.376,A -85,B 0,C 180,E1 25503.152,E2 25503.152} C_VEL
LIN {X 0,Y 538.531,Z 1066.78,A -85,B 0,C 180,E1 25502.252,E2 25502.252} C_VEL
LIN {X 0,Y 537.868,Z 1088.589,A -85,B 0,C 180,E1 25501.716,E2 25501.716} C_VEL
LIN {X 0,Y 537.098,Z 1110.239,A -85,B 0,C 180,E1 25500.978,E2 25500.978} C_VEL
LIN {X 0,Y 536.202,Z 1130.642,A -85,B 0,C 180,E1 25500.092,E2 25500.092} C_VEL
LIN {X 0,Y 535.18,Z 1150.67,A -85,B 0,C 180,E1 25499.005,E2 25499.005} C_VEL
LIN {X 0,Y 534.038,Z 1171.143,A -85,B 0,C 180,E1 25497.665,E2 25497.665} C_VEL
LIN {X 0,Y 532.934,Z 1190.448,A -85,B 0,C 180,E1 25496.16,E2 25496.16} C_VEL
LIN {X 0,Y 531.904,Z 1208.36,A -85,B 0,C 180,E1 25494.522,E2 25494.522} C_VEL
LIN {X 0,Y 530.911,Z 1225.21,A -85,B 0,C 180,E1 25492.71,E2 25492.71} C_VEL
LIN {X 0,Y 530.066,Z 1240.723,A -85,B 0,C 180,E1 25490.77,E2 25490.77} C_VEL
LIN {X 0,Y 529.382,Z 1254.758,A -85,B 0,C 180,E1 25488.728,E2 25488.728} C_VEL
LIN {X 0,Y 528.85,Z 1267.353,A -85,B 0,C 180,E1 25486.587,E2 25486.587} C_VEL
LIN {X 0,Y 528.452,Z 1278.363,A -85,B 0,C 180,E1 25484.35,E2 25484.35} C_VEL
LIN {X 0,Y 528.184,Z 1287.887,A -85,B 0,C 180,E1 25482.018,E2 25482.018} C_VEL
LIN {X 0,Y 528.038,Z 1295.247,A -85,B 0,C 180,E1 25479.812,E2 25479.812} C_VEL
LIN {X 0,Y 527.955,Z 1301.162,A -85,B 0,C 180,E1 25477.508,E2 25477.508} C_VEL
LIN {X 0,Y 527.913,Z 1305.623,A -85,B 0,C 180,E1 25475.107,E2 25475.107} C_VEL
LIN {X 0,Y 527.902,Z 1308.338,A -85,B 0,C 180,E1 25472.823,E2 25472.823} C_VEL
LIN {X 0,Y 527.895,Z 1309.395,A -85,B 0,C 180,E1 25470.543,E2 25470.543} C_VEL
LIN {X 0,Y 527.899,Z 1308.949,A -85,B 0,C 180,E1 25468.155,E2 25468.155} C_VEL
LIN {X 0,Y 527.907,Z 1306.992,A -85,B 0,C 180,E1 25465.873,E2 25465.873} C_VEL
LIN {X 0,Y 527.93,Z 1303.398,A -85,B 0,C 180,E1 25463.584,E2 25463.584} C_VEL
LIN {X 0,Y 527.988,Z 1298.281,A -85,B 0,C 180,E1 25461.287,E2 25461.287} C_VEL
LIN {X 0,Y 528.095,Z 1291.759,A -85,B 0,C 180,E1 25459.086,E2 25459.086} C_VEL
LIN {X 0,Y 528.307,Z 1283.141,A -85,B 0,C 180,E1 25456.762,E2 25456.762} C_VEL
LIN {X 0,Y 528.628,Z 1273.117,A -85,B 0,C 180,E1 25454.533,E2 25454.533} C_VEL
LIN {X 0,Y 529.079,Z 1261.635,A -85,B 0,C 180,E1 25452.401,E2 25452.401} C_VEL
LIN {X 0,Y 529.666,Z 1248.792,A -85,B 0,C 180,E1 25450.366,E2 25450.366} C_VEL
LIN {X 0,Y 530.404,Z 1234.658,A -85,B 0,C 180,E1 25448.434,E2 25448.434} C_VEL
LIN {X 0,Y 531.293,Z 1218.837,A -85,B 0,C 180,E1 25446.57,E2 25446.57} C_VEL
LIN {X 0,Y 532.239,Z 1202.066,A -85,B 0,C 180,E1 25444.878,E2 25444.878} C_VEL
LIN {X 0,Y 533.337,Z 1183.407,A -85,B 0,C 180,E1 25443.261,E2 25443.261} C_VEL
LIN {X 0,Y 534.444,Z 1164.557,A -85,B 0,C 180,E1 25441.872,E2 25441.872} C_VEL
LIN {X 0,Y 535.463,Z 1144.851,A -85,B 0,C 180,E1 25440.656,E2 25440.656} C_VEL
LIN {X 0,Y 536.464,Z 1125.003,A -85,B 0,C 180,E1 25439.647,E2 25439.647} C_VEL
LIN {X 0,Y 537.335,Z 1104.51,A -85,B 0,C 180,E1 25438.8,E2 25438.8} C_VEL
LIN {X 0,Y 538.057,Z 1083.394,A -85,B 0,C 180,E1 25438.14,E2 25438.14} C_VEL
LIN {X 0,Y 538.606,Z 1060.937,A -85,B 0,C 180,E1 25437.644,E2 25437.644} C_VEL
LIN {X 0,Y 540.945,Z 840.428,A -85,B 0,C 180,E1 25434.322,E2 25434.322} C_VEL
LIN {X 0,Y 541.51,Z 772.436,A -85,B 0,C 180,E1 25433.271,E2 25433.271} C_VEL
LIN {X 0,Y 539.274,Z 759.097,A -85,B 0,C 180,E1 25432.868,E2 25432.868} C_VEL
LIN {X 0,Y 540.424,Z 721.298,A -85,B 0,C 180,E1 25430.405,E2 25430.405} C_VEL
LIN {X 0,Y 541.016,Z 696.564,A -85,B 0,C 180,E1 25428.779,E2 25428.779} C_VEL
LIN {X 0,Y 528.591,Z 669.322,A -85,B 0,C 180,E1 25425.799,E2 25425.799} C_VEL
LIN {X 0,Y 528.511,Z 668.898,A -85,B 0,C 180,E1 25425.119,E2 25425.119} C_VEL
LIN {X 0,Y 528.51,Z 668.859,A -85,B 0,C 180,E1 25421.753,E2 25421.753} C_VEL
LIN {X 0,Y 528.524,Z 668.89,A -85,B 0,C 180,E1 25418.273,E2 25418.273} C_VEL
LIN {X 0,Y 528.52,Z 668.893,A -85,B 0,C 180,E1 25414.813,E2 25414.813} C_VEL
LIN {X 0,Y 528.509,Z 668.9,A -85,B 0,C 180,E1 25411.349,E2 25411.349} C_VEL
LIN {X 0,Y 528.509,Z 668.901,A -85,B 0,C 180,E1 25407.981,E2 25407.981} C_VEL
LIN {X 0,Y 528.509,Z 668.888,A -85,B 0,C 180,E1 25404.595,E2 25404.595} C_VEL
LIN {X 0,Y 528.52,Z 668.894,A -85,B 0,C 180,E1 25401.151,E2 25401.151} C_VEL
LIN {X 0,Y 528.518,Z 668.898,A -85,B 0,C 180,E1 25397.619,E2 25397.619} C_VEL
LIN {X 0,Y 528.513,Z 668.894,A -85,B 0,C 180,E1 25394.237,E2 25394.237} C_VEL
LIN {X 0,Y 528.508,Z 668.897,A -85,B 0,C 180,E1 25390.795,E2 25390.795} C_VEL
LIN {X 0,Y 528.517,Z 668.895,A -85,B 0,C 180,E1 25387.391,E2 25387.391} C_VEL
LIN {X 0,Y 528.518,Z 668.894,A -85,B 0,C 180,E1 25383.905,E2 25383.905} C_VEL
LIN {X 0,Y 528.522,Z 668.898,A -85,B 0,C 180,E1 25380.433,E2 25380.433} C_VEL
LIN {X 0,Y 528.516,Z 668.892,A -85,B 0,C 180,E1 25377.072,E2 25377.072} C_VEL
LIN {X 0,Y 528.509,Z 668.889,A -85,B 0,C 180,E1 25373.7,E2 25373.7} C_VEL
LIN {X 0,Y 528.524,Z 668.9,A -85,B 0,C 180,E1 25370.263,E2 25370.263} C_VEL
LIN {X 0,Y 528.516,Z 668.896,A -85,B 0,C 180,E1 25366.767,E2 25366.767} C_VEL
LIN {X 0,Y 528.523,Z 668.894,A -85,B 0,C 180,E1 25363.288,E2 25363.288} C_VEL
LIN {X 0,Y 528.526,Z 668.894,A -85,B 0,C 180,E1 25359.767,E2 25359.767} C_VEL
LIN {X 0,Y 528.509,Z 668.894,A -85,B 0,C 180,E1 25356.355,E2 25356.355} C_VEL
LIN {X 0,Y 528.52,Z 668.896,A -85,B 0,C 180,E1 25352.997,E2 25352.997} C_VEL
LIN {X 0,Y 528.507,Z 668.87,A -85,B 0,C 180,E1 25349.616,E2 25349.616} C_VEL
LIN {X 0,Y 528.524,Z 668.896,A -85,B 0,C 180,E1 25346.147,E2 25346.147} C_VEL
LIN {X 0,Y 528.517,Z 668.877,A -85,B 0,C 180,E1 25342.607,E2 25342.607} C_VEL
LIN {X 0,Y 528.519,Z 668.889,A -85,B 0,C 180,E1 25341.618,E2 25341.618} C_VEL
LIN {X 0,Y 527.502,Z 669.025,A -85,B 0,C 180,E1 25340.783,E2 25340.783} C_VEL
LIN {X 0,Y 521.085,Z 669.809,A -85,B 0,C 180,E1 25338.437,E2 25338.437} C_VEL
LIN {X 0,Y 520.569,Z 669.863,A -85,B 0,C 180,E1 25337.826,E2 25337.826} C_VEL
LIN {X 0,Y 520.584,Z 669.887,A -85,B 0,C 180,E1 25334.354,E2 25334.354} C_VEL
LIN {X 0,Y 520.583,Z 669.888,A -85,B 0,C 180,E1 25330.768,E2 25330.768} C_VEL
LIN {X 0,Y 520.613,Z 670.068,A -85,B 0,C 180,E1 25327.78,E2 25327.78} C_VEL
LIN {X 0,Y 520.827,Z 671.077,A -85,B 0,C 180,E1 25327.623,E2 25327.623} C_VEL
LIN {X 0,Y 522.78,Z 674.481,A -85,B 0,C 180,E1 25327.375,E2 25327.375} C_VEL
LIN {X 0,Y 534.406,Z 693.313,A -85,B 0,C 180,E1 25326.091,E2 25326.091} C_VEL
LIN {X 0,Y 531.865,Z 909.817,A -85,B 0,C 180,E1 25322.794,E2 25322.794} C_VEL
LIN {X 0,Y 531.315,Z 931.754,A -85,B 0,C 180,E1 25322.318,E2 25322.318} C_VEL
LIN {X 0,Y 530.51,Z 952.426,A -85,B 0,C 180,E1 25321.68,E2 25321.68} C_VEL
LIN {X 0,Y 529.569,Z 973.137,A -85,B 0,C 180,E1 25320.837,E2 25320.837} C_VEL
LIN {X 0,Y 528.518,Z 993.023,A -85,B 0,C 180,E1 25319.837,E2 25319.837} C_VEL
LIN {X 0,Y 527.336,Z 1012.886,A -85,B 0,C 180,E1 25318.613,E2 25318.613} C_VEL
LIN {X 0,Y 526.09,Z 1032.173,A -85,B 0,C 180,E1 25317.195,E2 25317.195} C_VEL
LIN {X 0,Y 524.923,Z 1050.396,A -85,B 0,C 180,E1 25315.618,E2 25315.618} C_VEL
LIN {X 0,Y 523.802,Z 1067.702,A -85,B 0,C 180,E1 25313.87,E2 25313.87} C_VEL
LIN {X 0,Y 522.794,Z 1083.38,A -85,B 0,C 180,E1 25312.015,E2 25312.015} C_VEL
LIN {X 0,Y 521.917,Z 1098.495,A -85,B 0,C 180,E1 25309.937,E2 25309.937} C_VEL
LIN {X 0,Y 521.224,Z 1112.027,A -85,B 0,C 180,E1 25307.758,E2 25307.758} C_VEL
LIN {X 0,Y 520.72,Z 1123.466,A -85,B 0,C 180,E1 25305.594,E2 25305.594} C_VEL
LIN {X 0,Y 520.358,Z 1133.419,A -85,B 0,C 180,E1 25303.331,E2 25303.331} C_VEL
LIN {X 0,Y 520.122,Z 1141.974,A -85,B 0,C 180,E1 25300.971,E2 25300.971} C_VEL
LIN {X 0,Y 519.995,Z 1148.762,A -85,B 0,C 180,E1 25298.626,E2 25298.626} C_VEL
LIN {X 0,Y 519.928,Z 1153.73,A -85,B 0,C 180,E1 25296.293,E2 25296.293} C_VEL
LIN {X 0,Y 519.901,Z 1157.288,A -85,B 0,C 180,E1 25293.859,E2 25293.859} C_VEL
LIN {X 0,Y 519.894,Z 1159.123,A -85,B 0,C 180,E1 25291.543,E2 25291.543} C_VEL
LIN {X 0,Y 519.9,Z 1159.36,A -85,B 0,C 180,E1 25289.229,E2 25289.229} C_VEL
LIN {X 0,Y 519.907,Z 1158.169,A -85,B 0,C 180,E1 25286.913,E2 25286.913} C_VEL
LIN {X 0,Y 519.917,Z 1155.528,A -85,B 0,C 180,E1 25284.704,E2 25284.704} C_VEL
LIN {X 0,Y 519.962,Z 1151.011,A -85,B 0,C 180,E1 25282.264,E2 25282.264} C_VEL
LIN {X 0,Y 520.051,Z 1145.368,A -85,B 0,C 180,E1 25280.036,E2 25280.036} C_VEL
LIN {X 0,Y 520.219,Z 1138.048,A -85,B 0,C 180,E1 25277.795,E2 25277.795} C_VEL
LIN {X 0,Y 520.514,Z 1128.896,A -85,B 0,C 180,E1 25275.498,E2 25275.498} C_VEL
LIN {X 0,Y 520.942,Z 1118.161,A -85,B 0,C 180,E1 25273.268,E2 25273.268} C_VEL
LIN {X 0,Y 521.533,Z 1105.737,A -85,B 0,C 180,E1 25271.096,E2 25271.096} C_VEL
LIN {X 0,Y 522.338,Z 1091.043,A -85,B 0,C 180,E1 25268.909,E2 25268.909} C_VEL
LIN {X 0,Y 523.252,Z 1076.107,A -85,B 0,C 180,E1 25266.998,E2 25266.998} C_VEL
LIN {X 0,Y 524.323,Z 1059.619,A -85,B 0,C 180,E1 25265.191,E2 25265.191} C_VEL
LIN {X 0,Y 525.441,Z 1042.281,A -85,B 0,C 180,E1 25263.56,E2 25263.56} C_VEL
LIN {X 0,Y 526.667,Z 1023.372,A -85,B 0,C 180,E1 25262.037,E2 25262.037} C_VEL
LIN {X 0,Y 527.922,Z 1003.488,A -85,B 0,C 180,E1 25260.688,E2 25260.688} C_VEL
LIN {X 0,Y 529.016,Z 983.473,A -85,B 0,C 180,E1 25259.568,E2 25259.568} C_VEL
LIN {X 0,Y 530.072,Z 962.783,A -85,B 0,C 180,E1 25258.628,E2 25258.628} C_VEL
LIN {X 0,Y 530.956,Z 942.151,A -85,B 0,C 180,E1 25257.885,E2 25257.885} C_VEL
LIN {X 0,Y 531.627,Z 920.578,A -85,B 0,C 180,E1 25257.325,E2 25257.325} C_VEL
LIN {X 0,Y 532.138,Z 891.253,A -85,B 0,C 180,E1 25256.825,E2 25256.825} C_VEL
LIN {X 0,Y 534.38,Z 693.27,A -85,B 0,C 180,E1 25253.817,E2 25253.817} C_VEL
LIN {X 0,Y 522.78,Z 674.474,A -85,B 0,C 180,E1 25252.535,E2 25252.535} C_VEL
LIN {X 0,Y 520.848,Z 671.143,A -85,B 0,C 180,E1 25252.293,E2 25252.293} C_VEL
LIN {X 0,Y 520.597,Z 669.957,A -85,B 0,C 180,E1 25252.079,E2 25252.079} C_VEL
LIN {X 0,Y 520.571,Z 669.877,A -85,B 0,C 180,E1 25248.647,E2 25248.647} C_VEL
LIN {X 0,Y 520.577,Z 669.891,A -85,B 0,C 180,E1 25245.181,E2 25245.181} C_VEL
LIN {X 0,Y 520.571,Z 669.863,A -85,B 0,C 180,E1 25241.796,E2 25241.796} C_VEL
LIN {X 0,Y 520.583,Z 669.877,A -85,B 0,C 180,E1 25238.343,E2 25238.343} C_VEL
LIN {X 0,Y 520.576,Z 669.885,A -85,B 0,C 180,E1 25234.781,E2 25234.781} C_VEL
LIN {X 0,Y 520.574,Z 669.87,A -85,B 0,C 180,E1 25231.366,E2 25231.366} C_VEL
LIN {X 0,Y 520.57,Z 669.883,A -85,B 0,C 180,E1 25227.933,E2 25227.933} C_VEL
LIN {X 0,Y 520.589,Z 669.882,A -85,B 0,C 180,E1 25224.446,E2 25224.446} C_VEL
LIN {X 0,Y 520.588,Z 669.882,A -85,B 0,C 180,E1 25220.931,E2 25220.931} C_VEL
LIN {X 0,Y 520.573,Z 669.884,A -85,B 0,C 180,E1 25217.435,E2 25217.435} C_VEL
LIN {X 0,Y 520.586,Z 669.889,A -85,B 0,C 180,E1 25214.005,E2 25214.005} C_VEL
LIN {X 0,Y 520.575,Z 669.88,A -85,B 0,C 180,E1 25210.514,E2 25210.514} C_VEL
LIN {X 0,Y 520.583,Z 669.877,A -85,B 0,C 180,E1 25206.95,E2 25206.95} C_VEL
LIN {X 0,Y 520.586,Z 669.889,A -85,B 0,C 180,E1 25203.414,E2 25203.414} C_VEL
LIN {X 0,Y 520.569,Z 669.886,A -85,B 0,C 180,E1 25200,E2 25200} C_VEL
LIN {X 0,Y 520.573,Z 669.886,A -85,B 0,C 180,E1 25196.587,E2 25196.587} C_VEL
LIN {X 0,Y 520.581,Z 669.885,A -85,B 0,C 180,E1 25193.161,E2 25193.161} C_VEL
LIN {X 0,Y 520.58,Z 669.884,A -85,B 0,C 180,E1 25189.599,E2 25189.599} C_VEL
LIN {X 0,Y 520.57,Z 669.877,A -85,B 0,C 180,E1 25186.109,E2 25186.109} C_VEL
LIN {X 0,Y 520.57,Z 669.887,A -85,B 0,C 180,E1 25182.68,E2 25182.68} C_VEL
LIN {X 0,Y 520.579,Z 669.884,A -85,B 0,C 180,E1 25179.187,E2 25179.187} C_VEL
LIN {X 0,Y 520.578,Z 669.875,A -85,B 0,C 180,E1 25175.61,E2 25175.61} C_VEL
LIN {X 0,Y 520.572,Z 669.888,A -85,B 0,C 180,E1 25172.178,E2 25172.178} C_VEL
LIN {X 0,Y 520.569,Z 669.89,A -85,B 0,C 180,E1 25168.763,E2 25168.763} C_VEL
LIN {X 0,Y 520.576,Z 669.879,A -85,B 0,C 180,E1 25165.288,E2 25165.288} C_VEL
LIN {X 0,Y 520.585,Z 669.878,A -85,B 0,C 180,E1 25161.769,E2 25161.769} C_VEL
LIN {X 0,Y 520.575,Z 669.845,A -85,B 0,C 180,E1 25158.342,E2 25158.342} C_VEL
LIN {X 0,Y 520.59,Z 670.001,A -85,B 0,C 180,E1 25154.973,E2 25154.973} C_VEL
LIN {X 0,Y 520.697,Z 670.612,A -85,B 0,C 180,E1 25154.806,E2 25154.806} C_VEL
LIN {X 0,Y 534.211,Z 700.352,A -85,B 0,C 180,E1 25151.494,E2 25151.494} C_VEL
LIN {X 0,Y 532.786,Z 748.474,A -85,B 0,C 180,E1 25148.331,E2 25148.331} C_VEL
LIN {X 0,Y 532.626,Z 759.497,A -85,B 0,C 180,E1 25147.652,E2 25147.652} C_VEL
LIN {X 0,Y 535.237,Z 776.065,A -85,B 0,C 180,E1 25147.172,E2 25147.172} C_VEL
LIN {X 0,Y 532.499,Z 1009.266,A -85,B 0,C 180,E1 25143.61,E2 25143.61} C_VEL
LIN {X 0,Y 531.763,Z 1066.779,A -85,B 0,C 180,E1 25142.714,E2 25142.714} C_VEL
LIN {X 0,Y 531.037,Z 1088.586,A -85,B 0,C 180,E1 25142.173,E2 25142.173} C_VEL
LIN {X 0,Y 530.185,Z 1110.236,A -85,B 0,C 180,E1 25141.428,E2 25141.428} C_VEL
LIN {X 0,Y 529.214,Z 1130.403,A -85,B 0,C 180,E1 25140.545,E2 25140.545} C_VEL
LIN {X 0,Y 528.051,Z 1150.835,A -85,B 0,C 180,E1 25139.425,E2 25139.425} C_VEL
LIN {X 0,Y 526.793,Z 1171.14,A -85,B 0,C 180,E1 25138.079,E2 25138.079} C_VEL
LIN {X 0,Y 525.569,Z 1190.445,A -85,B 0,C 180,E1 25136.555,E2 25136.555} C_VEL
LIN {X 0,Y 524.428,Z 1208.122,A -85,B 0,C 180,E1 25134.919,E2 25134.919} C_VEL
LIN {X 0,Y 523.33,Z 1224.703,A -85,B 0,C 180,E1 25133.117,E2 25133.117} C_VEL
LIN {X 0,Y 522.408,Z 1239.876,A -85,B 0,C 180,E1 25131.206,E2 25131.206} C_VEL
LIN {X 0,Y 521.629,Z 1254.052,A -85,B 0,C 180,E1 25129.133,E2 25129.133} C_VEL
LIN {X 0,Y 521.015,Z 1266.731,A -85,B 0,C 180,E1 25126.959,E2 25126.959} C_VEL
LIN {X 0,Y 520.562,Z 1277.333,A -85,B 0,C 180,E1 25124.8,E2 25124.8} C_VEL
LIN {X 0,Y 520.248,Z 1287.073,A -85,B 0,C 180,E1 25122.43,E2 25122.43} C_VEL
LIN {X 0,Y 520.066,Z 1294.937,A -85,B 0,C 180,E1 25120.076,E2 25120.076} C_VEL
LIN {X 0,Y 519.972,Z 1300.908,A -85,B 0,C 180,E1 25117.735,E2 25117.735} C_VEL
LIN {X 0,Y 519.921,Z 1305.463,A -85,B 0,C 180,E1 25115.296,E2 25115.296} C_VEL
LIN {X 0,Y 519.904,Z 1308.235,A -85,B 0,C 180,E1 25112.976,E2 25112.976} C_VEL
LIN {X 0,Y 519.896,Z 1309.373,A -85,B 0,C 180,E1 25110.661,E2 25110.661} C_VEL
LIN {X 0,Y 519.895,Z 1309.083,A -85,B 0,C 180,E1 25108.347,E2 25108.347} C_VEL
LIN {X 0,Y 519.899,Z 1307.333,A -85,B 0,C 180,E1 25106.141,E2 25106.141} C_VEL
LIN {X 0,Y 519.924,Z 1303.809,A -85,B 0,C 180,E1 25103.707,E2 25103.707} C_VEL
LIN {X 0,Y 519.992,Z 1298.873,A -85,B 0,C 180,E1 25101.374,E2 25101.374} C_VEL
LIN {X 0,Y 520.103,Z 1292.469,A -85,B 0,C 180,E1 25099.141,E2 25099.141} C_VEL
LIN {X 0,Y 520.334,Z 1284.057,A -85,B 0,C 180,E1 25096.782,E2 25096.782} C_VEL
LIN {X 0,Y 520.685,Z 1274.222,A -85,B 0,C 180,E1 25094.52,E2 25094.52} C_VEL
LIN {X 0,Y 521.175,Z 1262.919,A -85,B 0,C 180,E1 25092.356,E2 25092.356} C_VEL
LIN {X 0,Y 521.862,Z 1249.536,A -85,B 0,C 180,E1 25090.173,E2 25090.173} C_VEL
LIN {X 0,Y 522.684,Z 1235.583,A -85,B 0,C 180,E1 25088.217,E2 25088.217} C_VEL
LIN {X 0,Y 523.638,Z 1220.144,A -85,B 0,C 180,E1 25086.361,E2 25086.361} C_VEL
LIN {X 0,Y 524.74,Z 1202.917,A -85,B 0,C 180,E1 25084.578,E2 25084.578} C_VEL
LIN {X 0,Y 525.965,Z 1184.139,A -85,B 0,C 180,E1 25082.917,E2 25082.917} C_VEL
LIN {X 0,Y 527.197,Z 1165.446,A -85,B 0,C 180,E1 25081.512,E2 25081.512} C_VEL
LIN {X 0,Y 528.323,Z 1145.753,A -85,B 0,C 180,E1 25080.276,E2 25080.276} C_VEL
LIN {X 0,Y 529.466,Z 1125.339,A -85,B 0,C 180,E1 25079.22,E2 25079.22} C_VEL
LIN {X 0,Y 530.436,Z 1104.727,A -85,B 0,C 180,E1 25078.355,E2 25078.355} C_VEL
LIN {X 0,Y 531.236,Z 1083.651,A -85,B 0,C 180,E1 25077.689,E2 25077.689} C_VEL
LIN {X 0,Y 531.843,Z 1061.127,A -85,B 0,C 180,E1 25077.184,E2 25077.184} C_VEL
LIN {X 0,Y 534.433,Z 841.827,A -85,B 0,C 180,E1 25073.842,E2 25073.842} C_VEL
LIN {X 0,Y 535.081,Z 773.903,A -85,B 0,C 180,E1 25072.78,E2 25072.78} C_VEL
LIN {X 0,Y 532.522,Z 758.484,A -85,B 0,C 180,E1 25072.308,E2 25072.308} C_VEL
LIN {X 0,Y 533.964,Z 708.553,A -85,B 0,C 180,E1 25069.053,E2 25069.053} C_VEL
LIN {X 0,Y 534.162,Z 700.04,A -85,B 0,C 180,E1 25068.48,E2 25068.48} C_VEL
LIN {X 0,Y 521.428,Z 672.602,A -85,B 0,C 180,E1 25065.429,E2 25065.429} C_VEL
LIN {X 0,Y 520.606,Z 670.123,A -85,B 0,C 180,E1 25065.109,E2 25065.109} C_VEL
LIN {X 0,Y 520.565,Z 669.839,A -85,B 0,C 180,E1 25061.944,E2 25061.944} C_VEL
LIN {X 0,Y 520.572,Z 669.882,A -85,B 0,C 180,E1 25058.584,E2 25058.584} C_VEL
LIN {X 0,Y 520.585,Z 669.885,A -85,B 0,C 180,E1 25055.048,E2 25055.048} C_VEL
LIN {X 0,Y 520.575,Z 669.887,A -85,B 0,C 180,E1 25051.487,E2 25051.487} C_VEL
LIN {X 0,Y 520.571,Z 669.891,A -85,B 0,C 180,E1 25048.071,E2 25048.071} C_VEL
LIN {X 0,Y 520.57,Z 669.875,A -85,B 0,C 180,E1 25044.632,E2 25044.632} C_VEL
LIN {X 0,Y 520.581,Z 669.883,A -85,B 0,C 180,E1 25041.167,E2 25041.167} C_VEL
LIN {X 0,Y 520.581,Z 669.884,A -85,B 0,C 180,E1 25037.666,E2 25037.666} C_VEL
LIN {X 0,Y 520.574,Z 669.883,A -85,B 0,C 180,E1 25034.232,E2 25034.232} C_VEL
LIN {X 0,Y 520.57,Z 669.887,A -85,B 0,C 180,E1 25030.849,E2 25030.849} C_VEL
LIN {X 0,Y 520.577,Z 669.883,A -85,B 0,C 180,E1 25027.393,E2 25027.393} C_VEL
LIN {X 0,Y 520.581,Z 669.883,A -85,B 0,C 180,E1 25023.854,E2 25023.854} C_VEL
LIN {X 0,Y 520.577,Z 669.887,A -85,B 0,C 180,E1 25020.33,E2 25020.33} C_VEL
LIN {X 0,Y 520.576,Z 669.883,A -85,B 0,C 180,E1 25016.917,E2 25016.917} C_VEL
LIN {X 0,Y 520.57,Z 669.877,A -85,B 0,C 180,E1 25013.493,E2 25013.493} C_VEL
LIN {X 0,Y 520.588,Z 669.884,A -85,B 0,C 180,E1 25010.046,E2 25010.046} C_VEL
LIN {X 0,Y 520.583,Z 669.886,A -85,B 0,C 180,E1 25006.561,E2 25006.561} C_VEL
LIN {X 0,Y 520.576,Z 669.883,A -85,B 0,C 180,E1 25003.025,E2 25003.025} C_VEL
LIN {X 0,Y 520.585,Z 669.882,A -85,B 0,C 180,E1 24999.54,E2 24999.54} C_VEL
LIN {X 0,Y 520.572,Z 669.885,A -85,B 0,C 180,E1 24996.092,E2 24996.092} C_VEL
LIN {X 0,Y 520.587,Z 669.88,A -85,B 0,C 180,E1 24992.537,E2 24992.537} C_VEL
LIN {X 0,Y 520.583,Z 669.86,A -85,B 0,C 180,E1 24989.02,E2 24989.02} C_VEL
LIN {X 0,Y 520.571,Z 669.887,A -85,B 0,C 180,E1 24985.619,E2 24985.619} C_VEL
LIN {X 0,Y 520.571,Z 669.869,A -85,B 0,C 180,E1 24982.215,E2 24982.215} C_VEL
LIN {X 0,Y 520.573,Z 669.879,A -85,B 0,C 180,E1 24978.792,E2 24978.792} C_VEL
LIN {X 0,Y 520.569,Z 669.863,A -85,B 0,C 180,E1 24977.826,E2 24977.826} C_VEL
LIN {X 0,Y 519.603,Z 669.984,A -85,B 0,C 180,E1 24976.978,E2 24976.978} C_VEL
LIN {X 0,Y 513.088,Z 670.825,A -85,B 0,C 180,E1 24974.534,E2 24974.534} C_VEL
LIN {X 0,Y 512.636,Z 670.87,A -85,B 0,C 180,E1 24973.975,E2 24973.975} C_VEL
LIN {X 0,Y 512.64,Z 670.88,A -85,B 0,C 180,E1 24970.477,E2 24970.477} C_VEL
LIN {X 0,Y 512.669,Z 671.082,A -85,B 0,C 180,E1 24968.472,E2 24968.472} C_VEL
LIN {X 0,Y 513.038,Z 672.545,A -85,B 0,C 180,E1 24968.291,E2 24968.291} C_VEL
LIN {X 0,Y 515.109,Z 675.709,A -85,B 0,C 180,E1 24968.039,E2 24968.039} C_VEL
LIN {X 0,Y 526.788,Z 694.554,A -85,B 0,C 180,E1 24966.686,E2 24966.686} C_VEL
LIN {X 0,Y 527.936,Z 696.792,A -85,B 0,C 180,E1 24966.551,E2 24966.551} C_VEL
LIN {X 0,Y 525.057,Z 915.36,A -85,B 0,C 180,E1 24963.169,E2 24963.169} C_VEL
LIN {X 0,Y 524.329,Z 936.767,A -85,B 0,C 180,E1 24962.647,E2 24962.647} C_VEL
LIN {X 0,Y 523.387,Z 958.471,A -85,B 0,C 180,E1 24961.916,E2 24961.916} C_VEL
LIN {X 0,Y 522.362,Z 978.279,A -85,B 0,C 180,E1 24961.053,E2 24961.053} C_VEL
LIN {X 0,Y 521.129,Z 998.052,A -85,B 0,C 180,E1 24959.986,E2 24959.986} C_VEL
LIN {X 0,Y 519.818,Z 1018.128,A -85,B 0,C 180,E1 24958.678,E2 24958.678} C_VEL
LIN {X 0,Y 518.519,Z 1036.49,A -85,B 0,C 180,E1 24957.259,E2 24957.259} C_VEL
LIN {X 0,Y 517.232,Z 1054.051,A -85,B 0,C 180,E1 24955.658,E2 24955.658} C_VEL
LIN {X 0,Y 515.969,Z 1071.794,A -85,B 0,C 180,E1 24953.769,E2 24953.769} C_VEL
LIN {X 0,Y 514.905,Z 1087.332,A -85,B 0,C 180,E1 24951.844,E2 24951.844} C_VEL
LIN {X 0,Y 513.995,Z 1101.579,A -85,B 0,C 180,E1 24949.783,E2 24949.783} C_VEL
LIN {X 0,Y 513.282,Z 1113.946,A -85,B 0,C 180,E1 24947.69,E2 24947.69} C_VEL
LIN {X 0,Y 512.716,Z 1125.583,A -85,B 0,C 180,E1 24945.379,E2 24945.379} C_VEL
LIN {X 0,Y 512.354,Z 1135.256,A -85,B 0,C 180,E1 24943.083,E2 24943.083} C_VEL
LIN {X 0,Y 512.121,Z 1143.038,A -85,B 0,C 180,E1 24940.802,E2 24940.802} C_VEL
LIN {X 0,Y 511.987,Z 1149.537,A -85,B 0,C 180,E1 24938.422,E2 24938.422} C_VEL
LIN {X 0,Y 511.926,Z 1154.143,A -85,B 0,C 180,E1 24936.167,E2 24936.167} C_VEL
LIN {X 0,Y 511.9,Z 1157.402,A -85,B 0,C 180,E1 24933.808,E2 24933.808} C_VEL
LIN {X 0,Y 511.898,Z 1159.19,A -85,B 0,C 180,E1 24931.455,E2 24931.455} C_VEL
LIN {X 0,Y 511.904,Z 1159.337,A -85,B 0,C 180,E1 24929.105,E2 24929.105} C_VEL
LIN {X 0,Y 511.915,Z 1157.945,A -85,B 0,C 180,E1 24926.641,E2 24926.641} C_VEL
LIN {X 0,Y 511.93,Z 1155.208,A -85,B 0,C 180,E1 24924.396,E2 24924.396} C_VEL
LIN {X 0,Y 511.981,Z 1150.563,A -85,B 0,C 180,E1 24921.945,E2 24921.945} C_VEL
LIN {X 0,Y 512.089,Z 1144.731,A -85,B 0,C 180,E1 24919.652,E2 24919.652} C_VEL
LIN {X 0,Y 512.285,Z 1137.231,A -85,B 0,C 180,E1 24917.374,E2 24917.374} C_VEL
LIN {X 0,Y 512.638,Z 1127.533,A -85,B 0,C 180,E1 24914.966,E2 24914.966} C_VEL
LIN {X 0,Y 513.155,Z 1116.562,A -85,B 0,C 180,E1 24912.697,E2 24912.697} C_VEL
LIN {X 0,Y 513.83,Z 1104.32,A -85,B 0,C 180,E1 24910.565,E2 24910.565} C_VEL
LIN {X 0,Y 514.703,Z 1090.19,A -85,B 0,C 180,E1 24908.461,E2 24908.461} C_VEL
LIN {X 0,Y 515.764,Z 1074.581,A -85,B 0,C 180,E1 24906.463,E2 24906.463} C_VEL
LIN {X 0,Y 516.969,Z 1057.911,A -85,B 0,C 180,E1 24904.629,E2 24904.629} C_VEL
LIN {X 0,Y 518.26,Z 1040.071,A -85,B 0,C 180,E1 24902.961,E2 24902.961} C_VEL
LIN {X 0,Y 519.606,Z 1020.916,A -85,B 0,C 180,E1 24901.434,E2 24901.434} C_VEL
LIN {X 0,Y 520.928,Z 1001.591,A -85,B 0,C 180,E1 24900.134,E2 24900.134} C_VEL
LIN {X 0,Y 522.184,Z 981.188,A -85,B 0,C 180,E1 24898.999,E2 24898.999} C_VEL
LIN {X 0,Y 523.256,Z 961.278,A -85,B 0,C 180,E1 24898.107,E2 24898.107} C_VEL
LIN {X 0,Y 524.189,Z 940.45,A -85,B 0,C 180,E1 24897.367,E2 24897.367} C_VEL
LIN {X 0,Y 524.938,Z 919.244,A -85,B 0,C 180,E1 24896.823,E2 24896.823} C_VEL
LIN {X 0,Y 525.491,Z 887.383,A -85,B 0,C 180,E1 24896.289,E2 24896.289} C_VEL
LIN {X 0,Y 527.938,Z 696.385,A -85,B 0,C 180,E1 24893.352,E2 24893.352} C_VEL
LIN {X 0,Y 517.525,Z 679.632,A -85,B 0,C 180,E1 24892.158,E2 24892.158} C_VEL
LIN {X 0,Y 514.928,Z 675.531,A -85,B 0,C 180,E1 24891.851,E2 24891.851} C_VEL
LIN {X 0,Y 512.948,Z 672.272,A -85,B 0,C 180,E1 24891.602,E2 24891.602} C_VEL
LIN {X 0,Y 512.657,Z 670.96,A -85,B 0,C 180,E1 24891.385,E2 24891.385} C_VEL
LIN {X 0,Y 512.647,Z 670.85,A -85,B 0,C 180,E1 24887.829,E2 24887.829} C_VEL
LIN {X 0,Y 512.633,Z 670.874,A -85,B 0,C 180,E1 24884.288,E2 24884.288} C_VEL
LIN {X 0,Y 512.635,Z 670.875,A -85,B 0,C 180,E1 24880.798,E2 24880.798} C_VEL
LIN {X 0,Y 512.638,Z 670.849,A -85,B 0,C 180,E1 24877.274,E2 24877.274} C_VEL
LIN {X 0,Y 512.642,Z 670.875,A -85,B 0,C 180,E1 24873.77,E2 24873.77} C_VEL
LIN {X 0,Y 512.628,Z 670.842,A -85,B 0,C 180,E1 24870.343,E2 24870.343} C_VEL
LIN {X 0,Y 512.639,Z 670.875,A -85,B 0,C 180,E1 24866.904,E2 24866.904} C_VEL
LIN {X 0,Y 512.636,Z 670.871,A -85,B 0,C 180,E1 24863.446,E2 24863.446} C_VEL
LIN {X 0,Y 512.646,Z 670.871,A -85,B 0,C 180,E1 24859.939,E2 24859.939} C_VEL
LIN {X 0,Y 512.647,Z 670.872,A -85,B 0,C 180,E1 24856.428,E2 24856.428} C_VEL
LIN {X 0,Y 512.631,Z 670.874,A -85,B 0,C 180,E1 24852.962,E2 24852.962} C_VEL
LIN {X 0,Y 512.644,Z 670.88,A -85,B 0,C 180,E1 24849.43,E2 24849.43} C_VEL
LIN {X 0,Y 512.648,Z 670.866,A -85,B 0,C 180,E1 24845.922,E2 24845.922} C_VEL
LIN {X 0,Y 512.633,Z 670.865,A -85,B 0,C 180,E1 24842.348,E2 24842.348} C_VEL
LIN {X 0,Y 512.638,Z 670.877,A -85,B 0,C 180,E1 24838.883,E2 24838.883} C_VEL
LIN {X 0,Y 512.637,Z 670.874,A -85,B 0,C 180,E1 24835.414,E2 24835.414} C_VEL
LIN {X 0,Y 512.643,Z 670.87,A -85,B 0,C 180,E1 24831.815,E2 24831.815} C_VEL
LIN {X 0,Y 512.634,Z 670.865,A -85,B 0,C 180,E1 24828.262,E2 24828.262} C_VEL
LIN {X 0,Y 512.631,Z 670.872,A -85,B 0,C 180,E1 24824.849,E2 24824.849} C_VEL
LIN {X 0,Y 512.637,Z 670.856,A -85,B 0,C 180,E1 24821.345,E2 24821.345} C_VEL
LIN {X 0,Y 512.642,Z 670.88,A -85,B 0,C 180,E1 24817.767,E2 24817.767} C_VEL
LIN {X 0,Y 512.632,Z 670.868,A -85,B 0,C 180,E1 24814.218,E2 24814.218} C_VEL
LIN {X 0,Y 512.631,Z 670.86,A -85,B 0,C 180,E1 24810.817,E2 24810.817} C_VEL
LIN {X 0,Y 512.636,Z 670.875,A -85,B 0,C 180,E1 24807.411,E2 24807.411} C_VEL
LIN {X 0,Y 512.644,Z 670.877,A -85,B 0,C 180,E1 24803.846,E2 24803.846} C_VEL
LIN {X 0,Y 512.636,Z 670.879,A -85,B 0,C 180,E1 24800.373,E2 24800.373} C_VEL
LIN {X 0,Y 512.625,Z 670.815,A -85,B 0,C 180,E1 24796.948,E2 24796.948} C_VEL
LIN {X 0,Y 512.677,Z 671.152,A -85,B 0,C 180,E1 24795.551,E2 24795.551} C_VEL
LIN {X 0,Y 514.267,Z 674.86,A -85,B 0,C 180,E1 24795.064,E2 24795.064} C_VEL
LIN {X 0,Y 527.38,Z 703.992,A -85,B 0,C 180,E1 24791.789,E2 24791.789} C_VEL
LIN {X 0,Y 525.752,Z 752.054,A -85,B 0,C 180,E1 24788.591,E2 24788.591} C_VEL
LIN {X 0,Y 525.711,Z 758.051,A -85,B 0,C 180,E1 24788.234,E2 24788.234} C_VEL
LIN {X 0,Y 528.765,Z 777.587,A -85,B 0,C 180,E1 24787.662,E2 24787.662} C_VEL
LIN {X 0,Y 525.856,Z 1007.867,A -85,B 0,C 180,E1 24784.115,E2 24784.115} C_VEL
LIN {X 0,Y 525.029,Z 1066.779,A -85,B 0,C 180,E1 24783.187,E2 24783.187} C_VEL
LIN {X 0,Y 524.251,Z 1088.454,A -85,B 0,C 180,E1 24782.645,E2 24782.645} C_VEL
LIN {X 0,Y 523.305,Z 1110.233,A -85,B 0,C 180,E1 24781.889,E2 24781.889} C_VEL
LIN {X 0,Y 522.248,Z 1130.4,A -85,B 0,C 180,E1 24780.997,E2 24780.997} C_VEL
LIN {X 0,Y 521.018,Z 1149.765,A -85,B 0,C 180,E1 24779.93,E2 24779.93} C_VEL
LIN {X 0,Y 519.647,Z 1170.325,A -85,B 0,C 180,E1 24778.563,E2 24778.563} C_VEL
LIN {X 0,Y 518.336,Z 1189.107,A -85,B 0,C 180,E1 24777.079,E2 24777.079} C_VEL
LIN {X 0,Y 517.029,Z 1206.917,A -85,B 0,C 180,E1 24775.423,E2 24775.423} C_VEL
LIN {X 0,Y 515.867,Z 1223.183,A -85,B 0,C 180,E1 24773.653,E2 24773.653} C_VEL
LIN {X 0,Y 514.786,Z 1239.03,A -85,B 0,C 180,E1 24771.655,E2 24771.655} C_VEL
LIN {X 0,Y 513.942,Z 1252.634,A -85,B 0,C 180,E1 24769.667,E2 24769.667} C_VEL
LIN {X 0,Y 513.205,Z 1265.46,A -85,B 0,C 180,E1 24767.459,E2 24767.459} C_VEL
LIN {X 0,Y 512.66,Z 1276.817,A -85,B 0,C 180,E1 24765.149,E2 24765.149} C_VEL
LIN {X 0,Y 512.312,Z 1286.258,A -85,B 0,C 180,E1 24762.855,E2 24762.855} C_VEL
LIN {X 0,Y 512.096,Z 1293.883,A -85,B 0,C 180,E1 24760.575,E2 24760.575} C_VEL
LIN {X 0,Y 511.975,Z 1300.146,A -85,B 0,C 180,E1 24758.196,E2 24758.196} C_VEL
LIN {X 0,Y 511.925,Z 1304.823,A -85,B 0,C 180,E1 24755.829,E2 24755.829} C_VEL
LIN {X 0,Y 511.91,Z 1307.787,A -85,B 0,C 180,E1 24753.471,E2 24753.471} C_VEL
LIN {X 0,Y 511.909,Z 1309.305,A -85,B 0,C 180,E1 24751.007,E2 24751.007} C_VEL
LIN {X 0,Y 511.907,Z 1309.259,A -85,B 0,C 180,E1 24748.769,E2 24748.769} C_VEL
LIN {X 0,Y 511.905,Z 1307.673,A -85,B 0,C 180,E1 24746.417,E2 24746.417} C_VEL
LIN {X 0,Y 511.921,Z 1304.632,A -85,B 0,C 180,E1 24744.058,E2 24744.058} C_VEL
LIN {X 0,Y 511.975,Z 1300.145,A -85,B 0,C 180,E1 24741.804,E2 24741.804} C_VEL
LIN {X 0,Y 512.096,Z 1293.883,A -85,B 0,C 180,E1 24739.425,E2 24739.425} C_VEL
LIN {X 0,Y 512.312,Z 1286.256,A -85,B 0,C 180,E1 24737.145,E2 24737.145} C_VEL
LIN {X 0,Y 512.66,Z 1276.816,A -85,B 0,C 180,E1 24734.851,E2 24734.851} C_VEL
LIN {X 0,Y 513.205,Z 1265.46,A -85,B 0,C 180,E1 24732.541,E2 24732.541} C_VEL
LIN {X 0,Y 513.947,Z 1252.557,A -85,B 0,C 180,E1 24730.321,E2 24730.321} C_VEL
LIN {X 0,Y 514.847,Z 1238.179,A -85,B 0,C 180,E1 24728.228,E2 24728.228} C_VEL
LIN {X 0,Y 515.904,Z 1222.677,A -85,B 0,C 180,E1 24726.288,E2 24726.288} C_VEL
LIN {X 0,Y 517.111,Z 1205.709,A -85,B 0,C 180,E1 24724.458,E2 24724.458} C_VEL
LIN {X 0,Y 518.44,Z 1187.766,A -85,B 0,C 180,E1 24722.802,E2 24722.802} C_VEL
LIN {X 0,Y 519.709,Z 1169.518,A -85,B 0,C 180,E1 24721.378,E2 24721.378} C_VEL
LIN {X 0,Y 521.075,Z 1148.764,A -85,B 0,C 180,E1 24720.011,E2 24720.011} C_VEL
LIN {X 0,Y 522.32,Z 1129.176,A -85,B 0,C 180,E1 24718.944,E2 24718.944} C_VEL
LIN {X 0,Y 523.342,Z 1109.504,A -85,B 0,C 180,E1 24718.081,E2 24718.081} C_VEL
LIN {X 0,Y 524.308,Z 1087.168,A -85,B 0,C 180,E1 24717.319,E2 24717.319} C_VEL
LIN {X 0,Y 525.05,Z 1065.687,A -85,B 0,C 180,E1 24716.792,E2 24716.792} C_VEL
LIN {X 0,Y 526.935,Z 921.603,A -85,B 0,C 180,E1 24714.562,E2 24714.562} C_VEL
LIN {X 0,Y 528.612,Z 775.355,A -85,B 0,C 180,E1 24712.289,E2 24712.289} C_VEL
LIN {X 0,Y 525.608,Z 757.021,A -85,B 0,C 180,E1 24711.728,E2 24711.728} C_VEL
LIN {X 0,Y 527.24,Z 708.091,A -85,B 0,C 180,E1 24708.488,E2 24708.488} C_VEL
LIN {X 0,Y 527.301,Z 703.583,A -85,B 0,C 180,E1 24708.176,E2 24708.176} C_VEL
LIN {X 0,Y 514.125,Z 674.64,A -85,B 0,C 180,E1 24704.906,E2 24704.906} C_VEL
LIN {X 0,Y 512.667,Z 671.091,A -85,B 0,C 180,E1 24704.44,E2 24704.44} C_VEL
LIN {X 0,Y 512.643,Z 670.838,A -85,B 0,C 180,E1 24701.241,E2 24701.241} C_VEL
LIN {X 0,Y 512.63,Z 670.865,A -85,B 0,C 180,E1 24697.823,E2 24697.823} C_VEL
LIN {X 0,Y 512.631,Z 670.864,A -85,B 0,C 180,E1 24694.41,E2 24694.41} C_VEL
LIN {X 0,Y 512.637,Z 670.878,A -85,B 0,C 180,E1 24690.991,E2 24690.991} C_VEL
LIN {X 0,Y 512.645,Z 670.874,A -85,B 0,C 180,E1 24687.406,E2 24687.406} C_VEL
LIN {X 0,Y 512.632,Z 670.869,A -85,B 0,C 180,E1 24683.833,E2 24683.833} C_VEL
LIN {X 0,Y 512.631,Z 670.873,A -85,B 0,C 180,E1 24680.434,E2 24680.434} C_VEL
LIN {X 0,Y 512.64,Z 670.873,A -85,B 0,C 180,E1 24676.894,E2 24676.894} C_VEL
LIN {X 0,Y 512.638,Z 670.857,A -85,B 0,C 180,E1 24673.288,E2 24673.288} C_VEL
LIN {X 0,Y 512.633,Z 670.877,A -85,B 0,C 180,E1 24669.883,E2 24669.883} C_VEL
LIN {X 0,Y 512.631,Z 670.873,A -85,B 0,C 180,E1 24666.495,E2 24666.495} C_VEL
LIN {X 0,Y 512.643,Z 670.87,A -85,B 0,C 180,E1 24663.018,E2 24663.018} C_VEL
LIN {X 0,Y 512.647,Z 670.874,A -85,B 0,C 180,E1 24659.441,E2 24659.441} C_VEL
LIN {X 0,Y 512.633,Z 670.875,A -85,B 0,C 180,E1 24655.861,E2 24655.861} C_VEL
LIN {X 0,Y 512.652,Z 670.871,A -85,B 0,C 180,E1 24652.379,E2 24652.379} C_VEL
LIN {X 0,Y 512.642,Z 670.87,A -85,B 0,C 180,E1 24648.82,E2 24648.82} C_VEL
LIN {X 0,Y 512.643,Z 670.871,A -85,B 0,C 180,E1 24645.312,E2 24645.312} C_VEL
LIN {X 0,Y 512.648,Z 670.88,A -85,B 0,C 180,E1 24641.769,E2 24641.769} C_VEL
LIN {X 0,Y 512.635,Z 670.873,A -85,B 0,C 180,E1 24638.248,E2 24638.248} C_VEL
LIN {X 0,Y 512.647,Z 670.872,A -85,B 0,C 180,E1 24634.714,E2 24634.714} C_VEL
LIN {X 0,Y 512.646,Z 670.851,A -85,B 0,C 180,E1 24631.127,E2 24631.127} C_VEL
LIN {X 0,Y 512.631,Z 670.868,A -85,B 0,C 180,E1 24627.695,E2 24627.695} C_VEL
LIN {X 0,Y 512.636,Z 670.857,A -85,B 0,C 180,E1 24624.228,E2 24624.228} C_VEL
LIN {X 0,Y 512.649,Z 670.875,A -85,B 0,C 180,E1 24620.663,E2 24620.663} C_VEL
LIN {X 0,Y 512.632,Z 670.847,A -85,B 0,C 180,E1 24617.101,E2 24617.101} C_VEL
LIN {X 0,Y 512.636,Z 670.87,A -85,B 0,C 180,E1 24613.975,E2 24613.975} C_VEL
LIN {X 0,Y 511.634,Z 670.992,A -85,B 0,C 180,E1 24613.114,E2 24613.114} C_VEL
LIN {X 0,Y 505.145,Z 671.821,A -85,B 0,C 180,E1 24610.632,E2 24610.632} C_VEL
LIN {X 0,Y 504.709,Z 671.864,A -85,B 0,C 180,E1 24610.064,E2 24610.064} C_VEL
LIN {X 0,Y 504.734,Z 672.145,A -85,B 0,C 180,E1 24609.191,E2 24609.191} C_VEL
LIN {X 0,Y 505.178,Z 673.752,A -85,B 0,C 180,E1 24609.007,E2 24609.007} C_VEL
LIN {X 0,Y 507.326,Z 676.827,A -85,B 0,C 180,E1 24608.743,E2 24608.743} C_VEL
LIN {X 0,Y 520.641,Z 697.983,A -85,B 0,C 180,E1 24607.157,E2 24607.157} C_VEL
LIN {X 0,Y 521.569,Z 700.209,A -85,B 0,C 180,E1 24607.038,E2 24607.038} C_VEL
LIN {X 0,Y 518.355,Z 915.832,A -85,B 0,C 180,E1 24603.646,E2 24603.646} C_VEL
LIN {X 0,Y 517.561,Z 937.183,A -85,B 0,C 180,E1 24603.116,E2 24603.116} C_VEL
LIN {X 0,Y 516.507,Z 959.227,A -85,B 0,C 180,E1 24602.36,E2 24602.36} C_VEL
LIN {X 0,Y 515.367,Z 979.571,A -85,B 0,C 180,E1 24601.458,E2 24601.458} C_VEL
LIN {X 0,Y 513.976,Z 999.787,A -85,B 0,C 180,E1 24600.336,E2 24600.336} C_VEL
LIN {X 0,Y 512.527,Z 1019.759,A -85,B 0,C 180,E1 24598.997,E2 24598.997} C_VEL
LIN {X 0,Y 511.125,Z 1037.965,A -85,B 0,C 180,E1 24597.557,E2 24597.557} C_VEL
LIN {X 0,Y 509.693,Z 1055.751,A -85,B 0,C 180,E1 24595.892,E2 24595.892} C_VEL
LIN {X 0,Y 508.387,Z 1072.306,A -85,B 0,C 180,E1 24594.084,E2 24594.084} C_VEL
LIN {X 0,Y 507.207,Z 1087.869,A -85,B 0,C 180,E1 24592.117,E2 24592.117} C_VEL
LIN {X 0,Y 506.197,Z 1102.353,A -85,B 0,C 180,E1 24589.981,E2 24589.981} C_VEL
LIN {X 0,Y 505.416,Z 1114.585,A -85,B 0,C 180,E1 24587.856,E2 24587.856} C_VEL
LIN {X 0,Y 504.794,Z 1126.106,A -85,B 0,C 180,E1 24585.509,E2 24585.509} C_VEL
LIN {X 0,Y 504.396,Z 1135.695,A -85,B 0,C 180,E1 24583.177,E2 24583.177} C_VEL
LIN {X 0,Y 504.14,Z 1143.393,A -85,B 0,C 180,E1 24580.86,E2 24580.86} C_VEL
LIN {X 0,Y 503.989,Z 1150.047,A -85,B 0,C 180,E1 24578.327,E2 24578.327} C_VEL
LIN {X 0,Y 503.926,Z 1154.754,A -85,B 0,C 180,E1 24575.922,E2 24575.922} C_VEL
LIN {X 0,Y 503.906,Z 1157.744,A -85,B 0,C 180,E1 24573.526,E2 24573.526} C_VEL
LIN {X 0,Y 503.909,Z 1159.296,A -85,B 0,C 180,E1 24571.023,E2 24571.023} C_VEL
LIN {X 0,Y 503.906,Z 1159.246,A -85,B 0,C 180,E1 24568.636,E2 24568.636} C_VEL
LIN {X 0,Y 503.905,Z 1157.606,A -85,B 0,C 180,E1 24566.246,E2 24566.246} C_VEL
LIN {X 0,Y 503.929,Z 1154.51,A -85,B 0,C 180,E1 24563.85,E2 24563.85} C_VEL
LIN {X 0,Y 503.993,Z 1149.991,A -85,B 0,C 180,E1 24561.558,E2 24561.558} C_VEL
LIN {X 0,Y 504.145,Z 1143.313,A -85,B 0,C 180,E1 24559.025,E2 24559.025} C_VEL
LIN {X 0,Y 504.403,Z 1135.598,A -85,B 0,C 180,E1 24556.707,E2 24556.707} C_VEL
LIN {X 0,Y 504.807,Z 1125.982,A -85,B 0,C 180,E1 24554.374,E2 24554.374} C_VEL
LIN {X 0,Y 505.426,Z 1114.428,A -85,B 0,C 180,E1 24552.025,E2 24552.025} C_VEL
LIN {X 0,Y 506.208,Z 1102.161,A -85,B 0,C 180,E1 24549.899,E2 24549.899} C_VEL
LIN {X 0,Y 507.158,Z 1088.489,A -85,B 0,C 180,E1 24547.88,E2 24547.88} C_VEL
LIN {X 0,Y 508.356,Z 1072.687,A -85,B 0,C 180,E1 24545.87,E2 24545.87} C_VEL
LIN {X 0,Y 509.663,Z 1056.155,A -85,B 0,C 180,E1 24544.058,E2 24544.058} C_VEL
LIN {X 0,Y 511.101,Z 1038.241,A -85,B 0,C 180,E1 24542.379,E2 24542.379} C_VEL
LIN {X 0,Y 512.51,Z 1019.961,A -85,B 0,C 180,E1 24540.928,E2 24540.928} C_VEL
LIN {X 0,Y 513.996,Z 999.463,A -85,B 0,C 180,E1 24539.554,E2 24539.554} C_VEL
LIN {X 0,Y 515.339,Z 980.034,A -85,B 0,C 180,E1 24538.475,E2 24538.475} C_VEL
LIN {X 0,Y 516.483,Z 959.724,A -85,B 0,C 180,E1 24537.571,E2 24537.571} C_VEL
LIN {X 0,Y 517.564,Z 937.238,A -85,B 0,C 180,E1 24536.796,E2 24536.796} C_VEL
LIN {X 0,Y 518.355,Z 915.871,A -85,B 0,C 180,E1 24536.265,E2 24536.265} C_VEL
LIN {X 0,Y 521.533,Z 699.573,A -85,B 0,C 180,E1 24532.858,E2 24532.858} C_VEL
LIN {X 0,Y 512.24,Z 684.6,A -85,B 0,C 180,E1 24531.766,E2 24531.766} C_VEL
LIN {X 0,Y 506.968,Z 676.494,A -85,B 0,C 180,E1 24531.127,E2 24531.127} C_VEL
LIN {X 0,Y 505.005,Z 673.27,A -85,B 0,C 180,E1 24530.872,E2 24530.872} C_VEL
LIN {X 0,Y 504.707,Z 671.972,A -85,B 0,C 180,E1 24530.66,E2 24530.66} C_VEL
LIN {X 0,Y 504.699,Z 671.838,A -85,B 0,C 180,E1 24527.196,E2 24527.196} C_VEL
LIN {X 0,Y 504.703,Z 671.841,A -85,B 0,C 180,E1 24523.691,E2 24523.691} C_VEL
LIN {X 0,Y 504.697,Z 671.866,A -85,B 0,C 180,E1 24520.08,E2 24520.08} C_VEL
LIN {X 0,Y 504.691,Z 671.835,A -85,B 0,C 180,E1 24516.607,E2 24516.607} C_VEL
LIN {X 0,Y 504.705,Z 671.867,A -85,B 0,C 180,E1 24513.074,E2 24513.074} C_VEL
LIN {X 0,Y 504.705,Z 671.828,A -85,B 0,C 180,E1 24509.557,E2 24509.557} C_VEL
LIN {X 0,Y 504.696,Z 671.865,A -85,B 0,C 180,E1 24506.092,E2 24506.092} C_VEL
LIN {X 0,Y 504.706,Z 671.865,A -85,B 0,C 180,E1 24502.602,E2 24502.602} C_VEL
LIN {X 0,Y 504.7,Z 671.86,A -85,B 0,C 180,E1 24499.08,E2 24499.08} C_VEL
LIN {X 0,Y 504.704,Z 671.86,A -85,B 0,C 180,E1 24495.513,E2 24495.513} C_VEL
LIN {X 0,Y 504.708,Z 671.86,A -85,B 0,C 180,E1 24492.006,E2 24492.006} C_VEL
LIN {X 0,Y 504.693,Z 671.864,A -85,B 0,C 180,E1 24488.545,E2 24488.545} C_VEL
LIN {X 0,Y 504.704,Z 671.867,A -85,B 0,C 180,E1 24485.001,E2 24485.001} C_VEL
LIN {X 0,Y 504.71,Z 671.855,A -85,B 0,C 180,E1 24481.476,E2 24481.476} C_VEL
LIN {X 0,Y 504.694,Z 671.858,A -85,B 0,C 180,E1 24477.957,E2 24477.957} C_VEL
LIN {X 0,Y 504.697,Z 671.865,A -85,B 0,C 180,E1 24474.429,E2 24474.429} C_VEL
LIN {X 0,Y 504.701,Z 671.862,A -85,B 0,C 180,E1 24470.996,E2 24470.996} C_VEL
LIN {X 0,Y 504.698,Z 671.844,A -85,B 0,C 180,E1 24467.413,E2 24467.413} C_VEL
LIN {X 0,Y 504.694,Z 671.869,A -85,B 0,C 180,E1 24463.898,E2 24463.898} C_VEL
LIN {X 0,Y 504.692,Z 671.845,A -85,B 0,C 180,E1 24460.439,E2 24460.439} C_VEL
LIN {X 0,Y 504.708,Z 671.859,A -85,B 0,C 180,E1 24456.906,E2 24456.906} C_VEL
LIN {X 0,Y 504.696,Z 671.87,A -85,B 0,C 180,E1 24453.275,E2 24453.275} C_VEL
LIN {X 0,Y 504.692,Z 671.851,A -85,B 0,C 180,E1 24449.788,E2 24449.788} C_VEL
LIN {X 0,Y 504.698,Z 671.849,A -85,B 0,C 180,E1 24446.309,E2 24446.309} C_VEL
LIN {X 0,Y 504.702,Z 671.853,A -85,B 0,C 180,E1 24442.684,E2 24442.684} C_VEL
LIN {X 0,Y 504.697,Z 671.842,A -85,B 0,C 180,E1 24439.324,E2 24439.324} C_VEL
LIN {X 0,Y 504.729,Z 672.022,A -85,B 0,C 180,E1 24436.306,E2 24436.306} C_VEL
LIN {X 0,Y 504.942,Z 673.035,A -85,B 0,C 180,E1 24436.116,E2 24436.116} C_VEL
LIN {X 0,Y 513.442,Z 691.509,A -85,B 0,C 180,E1 24433.887,E2 24433.887} C_VEL
LIN {X 0,Y 520.563,Z 707.627,A -85,B 0,C 180,E1 24432.091,E2 24432.091} C_VEL
LIN {X 0,Y 518.772,Z 755.811,A -85,B 0,C 180,E1 24428.858,E2 24428.858} C_VEL
LIN {X 0,Y 522.312,Z 779.014,A -85,B 0,C 180,E1 24428.162,E2 24428.162} C_VEL
LIN {X 0,Y 519.2,Z 1010.793,A -85,B 0,C 180,E1 24424.566,E2 24424.566} C_VEL
LIN {X 0,Y 518.326,Z 1066.951,A -85,B 0,C 180,E1 24423.669,E2 24423.669} C_VEL
LIN {X 0,Y 517.504,Z 1088.322,A -85,B 0,C 180,E1 24423.129,E2 24423.129} C_VEL
LIN {X 0,Y 516.459,Z 1110.229,A -85,B 0,C 180,E1 24422.363,E2 24422.363} C_VEL
LIN {X 0,Y 515.316,Z 1130.398,A -85,B 0,C 180,E1 24421.461,E2 24421.461} C_VEL
LIN {X 0,Y 513.905,Z 1150.767,A -85,B 0,C 180,E1 24420.323,E2 24420.323} C_VEL
LIN {X 0,Y 512.479,Z 1170.321,A -85,B 0,C 180,E1 24419,E2 24419} C_VEL
LIN {X 0,Y 511.085,Z 1188.435,A -85,B 0,C 180,E1 24417.559,E2 24417.559} C_VEL
LIN {X 0,Y 509.65,Z 1206.295,A -85,B 0,C 180,E1 24415.883,E2 24415.883} C_VEL
LIN {X 0,Y 508.391,Z 1222.217,A -85,B 0,C 180,E1 24414.14,E2 24414.14} C_VEL
LIN {X 0,Y 507.25,Z 1237.33,A -85,B 0,C 180,E1 24412.237,E2 24412.237} C_VEL
LIN {X 0,Y 506.226,Z 1251.87,A -85,B 0,C 180,E1 24410.1,E2 24410.1} C_VEL
LIN {X 0,Y 505.42,Z 1264.538,A -85,B 0,C 180,E1 24407.909,E2 24407.909} C_VEL
LIN {X 0,Y 504.784,Z 1276.301,A -85,B 0,C 180,E1 24405.509,E2 24405.509} C_VEL
LIN {X 0,Y 504.385,Z 1285.851,A -85,B 0,C 180,E1 24403.177,E2 24403.177} C_VEL
LIN {X 0,Y 504.131,Z 1293.53,A -85,B 0,C 180,E1 24400.86,E2 24400.86} C_VEL
LIN {X 0,Y 503.986,Z 1299.892,A -85,B 0,C 180,E1 24398.442,E2 24398.442} C_VEL
LIN {X 0,Y 503.923,Z 1304.43,A -85,B 0,C 180,E1 24396.151,E2 24396.151} C_VEL
LIN {X 0,Y 503.9,Z 1307.561,A -85,B 0,C 180,E1 24393.754,E2 24393.754} C_VEL
LIN {X 0,Y 503.902,Z 1309.237,A -85,B 0,C 180,E1 24391.364,E2 24391.364} C_VEL
LIN {X 0,Y 503.905,Z 1309.327,A -85,B 0,C 180,E1 24389.09,E2 24389.09} C_VEL
LIN {X 0,Y 503.912,Z 1307.897,A -85,B 0,C 180,E1 24386.588,E2 24386.588} C_VEL
LIN {X 0,Y 503.926,Z 1304.981,A -85,B 0,C 180,E1 24384.192,E2 24384.192} C_VEL
LIN {X 0,Y 503.98,Z 1300.399,A -85,B 0,C 180,E1 24381.788,E2 24381.788} C_VEL
LIN {X 0,Y 504.113,Z 1294.236,A -85,B 0,C 180,E1 24379.371,E2 24379.371} C_VEL
LIN {X 0,Y 504.347,Z 1286.664,A -85,B 0,C 180,E1 24377.055,E2 24377.055} C_VEL
LIN {X 0,Y 504.731,Z 1277.329,A -85,B 0,C 180,E1 24374.724,E2 24374.724} C_VEL
LIN {X 0,Y 505.299,Z 1266.729,A -85,B 0,C 180,E1 24372.497,E2 24372.497} C_VEL
LIN {X 0,Y 506.083,Z 1254.055,A -85,B 0,C 180,E1 24370.255,E2 24370.255} C_VEL
LIN {X 0,Y 507.059,Z 1239.873,A -85,B 0,C 180,E1 24368.119,E2 24368.119} C_VEL
LIN {X 0,Y 508.282,Z 1223.674,A -85,B 0,C 180,E1 24366.032,E2 24366.032} C_VEL
LIN {X 0,Y 509.553,Z 1207.576,A -85,B 0,C 180,E1 24364.245,E2 24364.245} C_VEL
LIN {X 0,Y 510.975,Z 1189.772,A -85,B 0,C 180,E1 24362.561,E2 24362.561} C_VEL
LIN {X 0,Y 512.414,Z 1171.137,A -85,B 0,C 180,E1 24361.06,E2 24361.06} C_VEL
LIN {X 0,Y 513.846,Z 1151.776,A -85,B 0,C 180,E1 24359.738,E2 24359.738} C_VEL
LIN {X 0,Y 515.22,Z 1131.642,A -85,B 0,C 180,E1 24358.604,E2 24358.604} C_VEL
LIN {X 0,Y 516.422,Z 1110.981,A -85,B 0,C 180,E1 24357.667,E2 24357.667} C_VEL
LIN {X 0,Y 517.45,Z 1089.643,A -85,B 0,C 180,E1 24356.909,E2 24356.909} C_VEL
LIN {X 0,Y 518.261,Z 1068.584,A -85,B 0,C 180,E1 24356.368,E2 24356.368} C_VEL
LIN {X 0,Y 518.888,Z 1033.822,A -85,B 0,C 180,E1 24355.788,E2 24355.788} C_VEL
LIN {X 0,Y 521.808,Z 814.247,A -85,B 0,C 180,E1 24352.389,E2 24352.389} C_VEL
LIN {X 0,Y 522.167,Z 776.834,A -85,B 0,C 180,E1 24351.789,E2 24351.789} C_VEL
LIN {X 0,Y 518.756,Z 755.181,A -85,B 0,C 180,E1 24351.109,E2 24351.109} C_VEL
LIN {X 0,Y 520.563,Z 707.629,A -85,B 0,C 180,E1 24347.909,E2 24347.909} C_VEL
LIN {X 0,Y 509.539,Z 682.893,A -85,B 0,C 180,E1 24345.103,E2 24345.103} C_VEL
LIN {X 0,Y 504.768,Z 672.272,A -85,B 0,C 180,E1 24343.79,E2 24343.79} C_VEL
LIN {X 0,Y 504.69,Z 671.799,A -85,B 0,C 180,E1 24343.194,E2 24343.194} C_VEL
LIN {X 0,Y 504.695,Z 671.867,A -85,B 0,C 180,E1 24339.767,E2 24339.767} C_VEL
LIN {X 0,Y 504.703,Z 671.867,A -85,B 0,C 180,E1 24336.266,E2 24336.266} C_VEL
LIN {X 0,Y 504.701,Z 671.862,A -85,B 0,C 180,E1 24332.606,E2 24332.606} C_VEL
LIN {X 0,Y 504.692,Z 671.848,A -85,B 0,C 180,E1 24329.115,E2 24329.115} C_VEL
LIN {X 0,Y 504.696,Z 671.855,A -85,B 0,C 180,E1 24325.66,E2 24325.66} C_VEL
LIN {X 0,Y 504.711,Z 671.87,A -85,B 0,C 180,E1 24322.111,E2 24322.111} C_VEL
LIN {X 0,Y 504.696,Z 671.845,A -85,B 0,C 180,E1 24318.6,E2 24318.6} C_VEL
LIN {X 0,Y 504.692,Z 671.861,A -85,B 0,C 180,E1 24315.159,E2 24315.159} C_VEL
LIN {X 0,Y 504.696,Z 671.853,A -85,B 0,C 180,E1 24311.658,E2 24311.658} C_VEL
LIN {X 0,Y 504.706,Z 671.858,A -85,B 0,C 180,E1 24308.086,E2 24308.086} C_VEL
LIN {X 0,Y 504.696,Z 671.863,A -85,B 0,C 180,E1 24304.545,E2 24304.545} C_VEL
LIN {X 0,Y 504.702,Z 671.866,A -85,B 0,C 180,E1 24301.021,E2 24301.021} C_VEL
LIN {X 0,Y 504.698,Z 671.854,A -85,B 0,C 180,E1 24297.502,E2 24297.502} C_VEL
LIN {X 0,Y 504.7,Z 671.854,A -85,B 0,C 180,E1 24293.859,E2 24293.859} C_VEL
LIN {X 0,Y 504.705,Z 671.869,A -85,B 0,C 180,E1 24290.421,E2 24290.421} C_VEL
LIN {X 0,Y 504.694,Z 671.863,A -85,B 0,C 180,E1 24286.947,E2 24286.947} C_VEL
LIN {X 0,Y 504.708,Z 671.861,A -85,B 0,C 180,E1 24283.425,E2 24283.425} C_VEL
LIN {X 0,Y 504.71,Z 671.858,A -85,B 0,C 180,E1 24279.836,E2 24279.836} C_VEL
LIN {X 0,Y 504.694,Z 671.861,A -85,B 0,C 180,E1 24276.41,E2 24276.41} C_VEL
LIN {X 0,Y 504.703,Z 671.861,A -85,B 0,C 180,E1 24272.893,E2 24272.893} C_VEL
LIN {X 0,Y 504.702,Z 671.828,A -85,B 0,C 180,E1 24269.393,E2 24269.393} C_VEL
LIN {X 0,Y 504.698,Z 671.865,A -85,B 0,C 180,E1 24265.762,E2 24265.762} C_VEL
LIN {X 0,Y 504.693,Z 671.841,A -85,B 0,C 180,E1 24262.227,E2 24262.227} C_VEL
LIN {X 0,Y 504.7,Z 671.85,A -85,B 0,C 180,E1 24258.722,E2 24258.722} C_VEL
LIN {X 0,Y 504.704,Z 671.866,A -85,B 0,C 180,E1 24255.149,E2 24255.149} C_VEL
LIN {X 0,Y 504.69,Z 671.844,A -85,B 0,C 180,E1 24251.579,E2 24251.579} C_VEL
LIN {X 0,Y 504.709,Z 671.864,A -85,B 0,C 180,E1 24250.064,E2 24250.064} C_VEL
LIN {X 0,Y 504.942,Z 672.877,A -85,B 0,C 180,E1 24249.61,E2 24249.61} C_VEL
LIN {X 0,Y 505.695,Z 676.057,A -85,B 0,C 180,E1 24249.135,E2 24249.135} C_VEL
LIN {X 0,Y 507.016,Z 681.348,A -85,B 0,C 180,E1 24248.706,E2 24248.706} C_VEL
LIN {X 0,Y 511.963,Z 696.63,A -85,B 0,C 180,E1 24247.959,E2 24247.959} C_VEL
LIN {X 0,Y 513.404,Z 699.652,A -85,B 0,C 180,E1 24247.772,E2 24247.772} C_VEL
LIN {X 0,Y 515.248,Z 703.154,A -85,B 0,C 180,E1 24247.544,E2 24247.544} C_VEL
LIN {X 0,Y 511.729,Z 915.818,A -85,B 0,C 180,E1 24244.15,E2 24244.15} C_VEL
LIN {X 0,Y 510.874,Z 936.918,A -85,B 0,C 180,E1 24243.619,E2 24243.619} C_VEL
LIN {X 0,Y 509.741,Z 958.505,A -85,B 0,C 180,E1 24242.876,E2 24242.876} C_VEL
LIN {X 0,Y 508.548,Z 978.312,A -85,B 0,C 180,E1 24241.995,E2 24241.995} C_VEL
LIN {X 0,Y 507.093,Z 998.071,A -85,B 0,C 180,E1 24240.906,E2 24240.906} C_VEL
LIN {X 0,Y 505.601,Z 1017.333,A -85,B 0,C 180,E1 24239.629,E2 24239.629} C_VEL
LIN {X 0,Y 504.036,Z 1035.828,A -85,B 0,C 180,E1 24238.171,E2 24238.171} C_VEL
LIN {X 0,Y 502.51,Z 1053.341,A -85,B 0,C 180,E1 24236.543,E2 24236.543} C_VEL
LIN {X 0,Y 501.035,Z 1070.286,A -85,B 0,C 180,E1 24234.712,E2 24234.712} C_VEL
LIN {X 0,Y 499.72,Z 1086.165,A -85,B 0,C 180,E1 24232.715,E2 24232.715} C_VEL
LIN {X 0,Y 498.613,Z 1100.046,A -85,B 0,C 180,E1 24230.666,E2 24230.666} C_VEL
LIN {X 0,Y 497.683,Z 1113.317,A -85,B 0,C 180,E1 24228.385,E2 24228.385} C_VEL
LIN {X 0,Y 497,Z 1124.553,A -85,B 0,C 180,E1 24226.118,E2 24226.118} C_VEL
LIN {X 0,Y 496.509,Z 1134.343,A -85,B 0,C 180,E1 24223.746,E2 24223.746} C_VEL
LIN {X 0,Y 496.194,Z 1142.689,A -85,B 0,C 180,E1 24221.271,E2 24221.271} C_VEL
LIN {X 0,Y 496.024,Z 1149.285,A -85,B 0,C 180,E1 24218.812,E2 24218.812} C_VEL
LIN {X 0,Y 495.945,Z 1153.941,A -85,B 0,C 180,E1 24216.482,E2 24216.482} C_VEL
LIN {X 0,Y 495.903,Z 1157.403,A -85,B 0,C 180,E1 24213.931,E2 24213.931} C_VEL
LIN {X 0,Y 495.896,Z 1159.191,A -85,B 0,C 180,E1 24211.502,E2 24211.502} C_VEL
LIN {X 0,Y 495.905,Z 1159.336,A -85,B 0,C 180,E1 24209.076,E2 24209.076} C_VEL
LIN {X 0,Y 495.913,Z 1157.944,A -85,B 0,C 180,E1 24206.532,E2 24206.532} C_VEL
LIN {X 0,Y 495.932,Z 1155.205,A -85,B 0,C 180,E1 24204.215,E2 24204.215} C_VEL
LIN {X 0,Y 495.993,Z 1150.752,A -85,B 0,C 180,E1 24201.771,E2 24201.771} C_VEL
LIN {X 0,Y 496.136,Z 1144.726,A -85,B 0,C 180,E1 24199.315,E2 24199.315} C_VEL
LIN {X 0,Y 496.385,Z 1137.227,A -85,B 0,C 180,E1 24196.962,E2 24196.962} C_VEL
LIN {X 0,Y 496.826,Z 1127.525,A -85,B 0,C 180,E1 24194.475,E2 24194.475} C_VEL
LIN {X 0,Y 497.445,Z 1116.967,A -85,B 0,C 180,E1 24192.211,E2 24192.211} C_VEL
LIN {X 0,Y 498.327,Z 1104.033,A -85,B 0,C 180,E1 24189.886,E2 24189.886} C_VEL
LIN {X 0,Y 499.378,Z 1090.177,A -85,B 0,C 180,E1 24187.765,E2 24187.765} C_VEL
LIN {X 0,Y 500.679,Z 1074.567,A -85,B 0,C 180,E1 24185.709,E2 24185.709} C_VEL
LIN {X 0,Y 502.12,Z 1057.956,A -85,B 0,C 180,E1 24183.829,E2 24183.829} C_VEL
LIN {X 0,Y 503.651,Z 1040.238,A -85,B 0,C 180,E1 24182.128,E2 24182.128} C_VEL
LIN {X 0,Y 505.227,Z 1021.702,A -85,B 0,C 180,E1 24180.608,E2 24180.608} C_VEL
LIN {X 0,Y 506.783,Z 1002.468,A -85,B 0,C 180,E1 24179.271,E2 24179.271} C_VEL
LIN {X 0,Y 508.261,Z 982.285,A -85,B 0,C 180,E1 24178.117,E2 24178.117} C_VEL
LIN {X 0,Y 509.553,Z 961.975,A -85,B 0,C 180,E1 24177.177,E2 24177.177} C_VEL
LIN {X 0,Y 510.678,Z 941.05,A -85,B 0,C 180,E1 24176.412,E2 24176.412} C_VEL
LIN {X 0,Y 511.563,Z 920.304,A -85,B 0,C 180,E1 24175.859,E2 24175.859} C_VEL
LIN {X 0,Y 512.227,Z 890.235,A -85,B 0,C 180,E1 24175.331,E2 24175.331} C_VEL
LIN {X 0,Y 515.21,Z 702.674,A -85,B 0,C 180,E1 24172.354,E2 24172.354} C_VEL
LIN {X 0,Y 504.789,Z 686.159,A -85,B 0,C 180,E1 24171.095,E2 24171.095} C_VEL
LIN {X 0,Y 499.084,Z 677.554,A -85,B 0,C 180,E1 24170.381,E2 24170.381} C_VEL
LIN {X 0,Y 497.089,Z 674.301,A -85,B 0,C 180,E1 24170.114,E2 24170.114} C_VEL
LIN {X 0,Y 496.78,Z 672.934,A -85,B 0,C 180,E1 24169.873,E2 24169.873} C_VEL
LIN {X 0,Y 496.752,Z 672.837,A -85,B 0,C 180,E1 24166.341,E2 24166.341} C_VEL
LIN {X 0,Y 496.757,Z 672.819,A -85,B 0,C 180,E1 24162.869,E2 24162.869} C_VEL
LIN {X 0,Y 496.771,Z 672.854,A -85,B 0,C 180,E1 24159.346,E2 24159.346} C_VEL
LIN {X 0,Y 496.755,Z 672.832,A -85,B 0,C 180,E1 24155.712,E2 24155.712} C_VEL
LIN {X 0,Y 496.754,Z 672.845,A -85,B 0,C 180,E1 24152.235,E2 24152.235} C_VEL
LIN {X 0,Y 496.77,Z 672.826,A -85,B 0,C 180,E1 24148.656,E2 24148.656} C_VEL
LIN {X 0,Y 496.765,Z 672.851,A -85,B 0,C 180,E1 24145.082,E2 24145.082} C_VEL
LIN {X 0,Y 496.754,Z 672.85,A -85,B 0,C 180,E1 24141.584,E2 24141.584} C_VEL
LIN {X 0,Y 496.772,Z 672.857,A -85,B 0,C 180,E1 24138.057,E2 24138.057} C_VEL
LIN {X 0,Y 496.772,Z 672.849,A -85,B 0,C 180,E1 24134.453,E2 24134.453} C_VEL
LIN {X 0,Y 496.755,Z 672.847,A -85,B 0,C 180,E1 24130.906,E2 24130.906} C_VEL
LIN {X 0,Y 496.763,Z 672.846,A -85,B 0,C 180,E1 24127.401,E2 24127.401} C_VEL
LIN {X 0,Y 496.767,Z 672.854,A -85,B 0,C 180,E1 24123.809,E2 24123.809} C_VEL
LIN {X 0,Y 496.757,Z 672.853,A -85,B 0,C 180,E1 24120.231,E2 24120.231} C_VEL
LIN {X 0,Y 496.757,Z 672.849,A -85,B 0,C 180,E1 24116.663,E2 24116.663} C_VEL
LIN {X 0,Y 496.764,Z 672.85,A -85,B 0,C 180,E1 24113.18,E2 24113.18} C_VEL
LIN {X 0,Y 496.762,Z 672.851,A -85,B 0,C 180,E1 24109.564,E2 24109.564} C_VEL
LIN {X 0,Y 496.753,Z 672.839,A -85,B 0,C 180,E1 24106.023,E2 24106.023} C_VEL
LIN {X 0,Y 496.757,Z 672.853,A -85,B 0,C 180,E1 24102.548,E2 24102.548} C_VEL
LIN {X 0,Y 496.767,Z 672.85,A -85,B 0,C 180,E1 24098.883,E2 24098.883} C_VEL
LIN {X 0,Y 496.754,Z 672.837,A -85,B 0,C 180,E1 24095.377,E2 24095.377} C_VEL
LIN {X 0,Y 496.756,Z 672.852,A -85,B 0,C 180,E1 24091.832,E2 24091.832} C_VEL
LIN {X 0,Y 496.765,Z 672.854,A -85,B 0,C 180,E1 24088.31,E2 24088.31} C_VEL
LIN {X 0,Y 496.758,Z 672.855,A -85,B 0,C 180,E1 24084.714,E2 24084.714} C_VEL
LIN {X 0,Y 496.756,Z 672.852,A -85,B 0,C 180,E1 24081.162,E2 24081.162} C_VEL
LIN {X 0,Y 496.755,Z 672.784,A -85,B 0,C 180,E1 24077.618,E2 24077.618} C_VEL
LIN {X 0,Y 496.822,Z 673.265,A -85,B 0,C 180,E1 24076.946,E2 24076.946} C_VEL
LIN {X 0,Y 506.03,Z 693.505,A -85,B 0,C 180,E1 24074.416,E2 24074.416} C_VEL
LIN {X 0,Y 513.774,Z 710.856,A -85,B 0,C 180,E1 24072.43,E2 24072.43} C_VEL
LIN {X 0,Y 512.014,Z 754.732,A -85,B 0,C 180,E1 24069.459,E2 24069.459} C_VEL
LIN {X 0,Y 515.9,Z 780.446,A -85,B 0,C 180,E1 24068.674,E2 24068.674} C_VEL
LIN {X 0,Y 512.523,Z 1012.954,A -85,B 0,C 180,E1 24065.031,E2 24065.031} C_VEL
LIN {X 0,Y 511.647,Z 1066.898,A -85,B 0,C 180,E1 24064.164,E2 24064.164} C_VEL
LIN {X 0,Y 510.822,Z 1087.656,A -85,B 0,C 180,E1 24063.641,E2 24063.641} C_VEL
LIN {X 0,Y 509.695,Z 1109.411,A -85,B 0,C 180,E1 24062.883,E2 24062.883} C_VEL
LIN {X 0,Y 508.5,Z 1129.182,A -85,B 0,C 180,E1 24061.999,E2 24061.999} C_VEL
LIN {X 0,Y 507.029,Z 1148.754,A -85,B 0,C 180,E1 24060.91,E2 24060.91} C_VEL
LIN {X 0,Y 505.412,Z 1169.507,A -85,B 0,C 180,E1 24059.51,E2 24059.51} C_VEL
LIN {X 0,Y 503.869,Z 1187.762,A -85,B 0,C 180,E1 24058.052,E2 24058.052} C_VEL
LIN {X 0,Y 502.311,Z 1205.708,A -85,B 0,C 180,E1 24056.351,E2 24056.351} C_VEL
LIN {X 0,Y 500.871,Z 1222.168,A -85,B 0,C 180,E1 24054.532,E2 24054.532} C_VEL
LIN {X 0,Y 499.617,Z 1237.331,A -85,B 0,C 180,E1 24052.596,E2 24052.596} C_VEL
LIN {X 0,Y 498.485,Z 1251.868,A -85,B 0,C 180,E1 24050.426,E2 24050.426} C_VEL
LIN {X 0,Y 497.622,Z 1264.187,A -85,B 0,C 180,E1 24048.266,E2 24048.266} C_VEL
LIN {X 0,Y 496.927,Z 1275.784,A -85,B 0,C 180,E1 24045.881,E2 24045.881} C_VEL
LIN {X 0,Y 496.472,Z 1285.431,A -85,B 0,C 180,E1 24043.51,E2 24043.51} C_VEL
LIN {X 0,Y 496.166,Z 1293.42,A -85,B 0,C 180,E1 24041.073,E2 24041.073} C_VEL
LIN {X 0,Y 496,Z 1299.892,A -85,B 0,C 180,E1 24038.579,E2 24038.579} C_VEL
LIN {X 0,Y 495.928,Z 1304.43,A -85,B 0,C 180,E1 24036.25,E2 24036.25} C_VEL
LIN {X 0,Y 495.9,Z 1307.56,A -85,B 0,C 180,E1 24033.815,E2 24033.815} C_VEL
LIN {X 0,Y 495.901,Z 1309.237,A -85,B 0,C 180,E1 24031.386,E2 24031.386} C_VEL
LIN {X 0,Y 495.905,Z 1309.327,A -85,B 0,C 180,E1 24029.076,E2 24029.076} C_VEL
LIN {X 0,Y 495.91,Z 1307.898,A -85,B 0,C 180,E1 24026.532,E2 24026.532} C_VEL
LIN {X 0,Y 495.928,Z 1305.14,A -85,B 0,C 180,E1 24024.215,E2 24024.215} C_VEL
LIN {X 0,Y 495.985,Z 1300.653,A -85,B 0,C 180,E1 24021.771,E2 24021.771} C_VEL
LIN {X 0,Y 496.123,Z 1294.937,A -85,B 0,C 180,E1 24019.433,E2 24019.433} C_VEL
LIN {X 0,Y 496.368,Z 1287.479,A -85,B 0,C 180,E1 24017.08,E2 24017.08} C_VEL
LIN {X 0,Y 496.808,Z 1277.79,A -85,B 0,C 180,E1 24014.582,E2 24014.582} C_VEL
LIN {X 0,Y 497.429,Z 1267.29,A -85,B 0,C 180,E1 24012.319,E2 24012.319} C_VEL
LIN {X 0,Y 498.274,Z 1254.764,A -85,B 0,C 180,E1 24010.055,E2 24010.055} C_VEL
LIN {X 0,Y 499.339,Z 1240.717,A -85,B 0,C 180,E1 24007.887,E2 24007.887} C_VEL
LIN {X 0,Y 500.628,Z 1225.209,A -85,B 0,C 180,E1 24005.832,E2 24005.832} C_VEL
LIN {X 0,Y 501.996,Z 1209.251,A -85,B 0,C 180,E1 24004.013,E2 24004.013} C_VEL
LIN {X 0,Y 503.517,Z 1191.773,A -85,B 0,C 180,E1 24002.312,E2 24002.312} C_VEL
LIN {X 0,Y 505.135,Z 1172.756,A -85,B 0,C 180,E1 24000.732,E2 24000.732} C_VEL
LIN {X 0,Y 506.688,Z 1153.761,A -85,B 0,C 180,E1 23999.396,E2 23999.396} C_VEL
LIN {X 0,Y 508.144,Z 1133.786,A -85,B 0,C 180,E1 23998.242,E2 23998.242} C_VEL
LIN {X 0,Y 509.529,Z 1112.458,A -85,B 0,C 180,E1 23997.242,E2 23997.242} C_VEL
LIN {X 0,Y 510.647,Z 1091.596,A -85,B 0,C 180,E1 23996.473,E2 23996.473} C_VEL
LIN {X 0,Y 511.479,Z 1071.021,A -85,B 0,C 180,E1 23995.929,E2 23995.929} C_VEL
LIN {X 0,Y 512.133,Z 1041.284,A -85,B 0,C 180,E1 23995.407,E2 23995.407} C_VEL
LIN {X 0,Y 515.308,Z 818.49,A -85,B 0,C 180,E1 23991.927,E2 23991.927} C_VEL
LIN {X 0,Y 515.739,Z 778.171,A -85,B 0,C 180,E1 23991.273,E2 23991.273} C_VEL
LIN {X 0,Y 511.949,Z 753.521,A -85,B 0,C 180,E1 23990.484,E2 23990.484} C_VEL
LIN {X 0,Y 513.774,Z 710.859,A -85,B 0,C 180,E1 23987.57,E2 23987.57} C_VEL
LIN {X 0,Y 502.025,Z 684.561,A -85,B 0,C 180,E1 23984.512,E2 23984.512} C_VEL
LIN {X 0,Y 496.814,Z 673.224,A -85,B 0,C 180,E1 23983.055,E2 23983.055} C_VEL
LIN {X 0,Y 496.756,Z 672.783,A -85,B 0,C 180,E1 23982.398,E2 23982.398} C_VEL
LIN {X 0,Y 496.754,Z 672.851,A -85,B 0,C 180,E1 23978.838,E2 23978.838} C_VEL
LIN {X 0,Y 496.758,Z 672.855,A -85,B 0,C 180,E1 23975.286,E2 23975.286} C_VEL
LIN {X 0,Y 496.765,Z 672.854,A -85,B 0,C 180,E1 23971.64,E2 23971.64} C_VEL
LIN {X 0,Y 496.755,Z 672.854,A -85,B 0,C 180,E1 23968.098,E2 23968.098} C_VEL
LIN {X 0,Y 496.756,Z 672.837,A -85,B 0,C 180,E1 23964.53,E2 23964.53} C_VEL
LIN {X 0,Y 496.767,Z 672.85,A -85,B 0,C 180,E1 23960.952,E2 23960.952} C_VEL
LIN {X 0,Y 496.754,Z 672.855,A -85,B 0,C 180,E1 23957.331,E2 23957.331} C_VEL
LIN {X 0,Y 496.754,Z 672.838,A -85,B 0,C 180,E1 23953.858,E2 23953.858} C_VEL
LIN {X 0,Y 496.765,Z 672.851,A -85,B 0,C 180,E1 23950.319,E2 23950.319} C_VEL
LIN {X 0,Y 496.759,Z 672.852,A -85,B 0,C 180,E1 23946.704,E2 23946.704} C_VEL
LIN {X 0,Y 496.758,Z 672.848,A -85,B 0,C 180,E1 23943.231,E2 23943.231} C_VEL
LIN {X 0,Y 496.762,Z 672.852,A -85,B 0,C 180,E1 23939.654,E2 23939.654} C_VEL
LIN {X 0,Y 496.764,Z 672.854,A -85,B 0,C 180,E1 23936.076,E2 23936.076} C_VEL
LIN {X 0,Y 496.77,Z 672.846,A -85,B 0,C 180,E1 23932.482,E2 23932.482} C_VEL
LIN {X 0,Y 496.763,Z 672.846,A -85,B 0,C 180,E1 23928.859,E2 23928.859} C_VEL
LIN {X 0,Y 496.761,Z 672.849,A -85,B 0,C 180,E1 23925.189,E2 23925.189} C_VEL
LIN {X 0,Y 496.77,Z 672.856,A -85,B 0,C 180,E1 23921.7,E2 23921.7} C_VEL
LIN {X 0,Y 496.764,Z 672.851,A -85,B 0,C 180,E1 23918.101,E2 23918.101} C_VEL
LIN {X 0,Y 496.763,Z 672.85,A -85,B 0,C 180,E1 23914.486,E2 23914.486} C_VEL
LIN {X 0,Y 496.763,Z 672.822,A -85,B 0,C 180,E1 23910.983,E2 23910.983} C_VEL
LIN {X 0,Y 496.756,Z 672.847,A -85,B 0,C 180,E1 23907.492,E2 23907.492} C_VEL
LIN {X 0,Y 496.764,Z 672.825,A -85,B 0,C 180,E1 23903.862,E2 23903.862} C_VEL
LIN {X 0,Y 496.758,Z 672.859,A -85,B 0,C 180,E1 23900.251,E2 23900.251} C_VEL
LIN {X 0,Y 496.752,Z 672.823,A -85,B 0,C 180,E1 23896.77,E2 23896.77} C_VEL
LIN {X 0,Y 496.762,Z 672.829,A -85,B 0,C 180,E1 23893.229,E2 23893.229} C_VEL
LIN {X 0,Y 496.803,Z 673.08,A -85,B 0,C 180,E1 23889.978,E2 23889.978} C_VEL
LIN {X 0,Y 497.17,Z 674.545,A -85,B 0,C 180,E1 23889.781,E2 23889.781} C_VEL
LIN {X 0,Y 499.084,Z 677.557,A -85,B 0,C 180,E1 23889.529,E2 23889.529} C_VEL
LIN {X 0,Y 500.524,Z 679.753,A -85,B 0,C 180,E1 23889.346,E2 23889.346} C_VEL
LIN {X 0,Y 511.166,Z 695.997,A -85,B 0,C 180,E1 23888.04,E2 23888.04} C_VEL
LIN {X 0,Y 513.404,Z 699.652,A -85,B 0,C 180,E1 23887.772,E2 23887.772} C_VEL
LIN {X 0,Y 514.127,Z 702.876,A -85,B 0,C 180,E1 23887.649,E2 23887.649} C_VEL
LIN {X 0,Y 513.335,Z 707.932,A -85,B 0,C 180,E1 23887.632,E2 23887.632} C_VEL
LIN {X 0,Y 509.058,Z 719.978,A -85,B 0,C 180,E1 23887.807,E2 23887.807} C_VEL
LIN {X 0,Y 508.656,Z 723.177,A -85,B 0,C 180,E1 23887.787,E2 23887.787} C_VEL
LIN {X 0,Y 505.201,Z 917.254,A -85,B 0,C 180,E1 23884.653,E2 23884.653} C_VEL
LIN {X 0,Y 504.323,Z 938.167,A -85,B 0,C 180,E1 23884.12,E2 23884.12} C_VEL
LIN {X 0,Y 503.144,Z 958.814,A -85,B 0,C 180,E1 23883.397,E2 23883.397} C_VEL
LIN {X 0,Y 501.758,Z 978.817,A -85,B 0,C 180,E1 23882.481,E2 23882.481} C_VEL
LIN {X 0,Y 499.966,Z 1000.089,A -85,B 0,C 180,E1 23881.262,E2 23881.262} C_VEL
LIN {X 0,Y 498.28,Z 1019.839,A -85,B 0,C 180,E1 23879.904,E2 23879.904} C_VEL
LIN {X 0,Y 496.625,Z 1037.978,A -85,B 0,C 180,E1 23878.433,E2 23878.433} C_VEL
LIN {X 0,Y 494.935,Z 1055.831,A -85,B 0,C 180,E1 23876.717,E2 23876.717} C_VEL
LIN {X 0,Y 493.361,Z 1072.318,A -85,B 0,C 180,E1 23874.867,E2 23874.867} C_VEL
LIN {X 0,Y 491.951,Z 1087.882,A -85,B 0,C 180,E1 23872.841,E2 23872.841} C_VEL
LIN {X 0,Y 490.726,Z 1102.361,A -85,B 0,C 180,E1 23870.639,E2 23870.639} C_VEL
LIN {X 0,Y 489.786,Z 1114.59,A -85,B 0,C 180,E1 23868.446,E2 23868.446} C_VEL
LIN {X 0,Y 489.025,Z 1126.111,A -85,B 0,C 180,E1 23866.022,E2 23866.022} C_VEL
LIN {X 0,Y 488.523,Z 1135.702,A -85,B 0,C 180,E1 23863.613,E2 23863.613} C_VEL
LIN {X 0,Y 488.2,Z 1143.508,A -85,B 0,C 180,E1 23861.181,E2 23861.181} C_VEL
LIN {X 0,Y 488.014,Z 1150.05,A -85,B 0,C 180,E1 23858.601,E2 23858.601} C_VEL
LIN {X 0,Y 487.93,Z 1154.756,A -85,B 0,C 180,E1 23856.117,E2 23856.117} C_VEL
LIN {X 0,Y 487.903,Z 1157.771,A -85,B 0,C 180,E1 23853.615,E2 23853.615} C_VEL
LIN {X 0,Y 487.909,Z 1159.295,A -85,B 0,C 180,E1 23851.057,E2 23851.057} C_VEL
LIN {X 0,Y 487.907,Z 1159.267,A -85,B 0,C 180,E1 23848.708,E2 23848.708} C_VEL
LIN {X 0,Y 487.906,Z 1157.718,A -85,B 0,C 180,E1 23846.24,E2 23846.24} C_VEL
LIN {X 0,Y 487.934,Z 1154.712,A -85,B 0,C 180,E1 23843.765,E2 23843.765} C_VEL
LIN {X 0,Y 488.019,Z 1149.988,A -85,B 0,C 180,E1 23841.28,E2 23841.28} C_VEL
LIN {X 0,Y 488.206,Z 1143.308,A -85,B 0,C 180,E1 23838.662,E2 23838.662} C_VEL
LIN {X 0,Y 488.529,Z 1135.593,A -85,B 0,C 180,E1 23836.266,E2 23836.266} C_VEL
LIN {X 0,Y 489.033,Z 1125.974,A -85,B 0,C 180,E1 23833.856,E2 23833.856} C_VEL
LIN {X 0,Y 489.799,Z 1114.418,A -85,B 0,C 180,E1 23831.431,E2 23831.431} C_VEL
LIN {X 0,Y 490.743,Z 1102.148,A -85,B 0,C 180,E1 23829.237,E2 23829.237} C_VEL
LIN {X 0,Y 491.893,Z 1088.476,A -85,B 0,C 180,E1 23827.156,E2 23827.156} C_VEL
LIN {X 0,Y 493.32,Z 1072.783,A -85,B 0,C 180,E1 23825.099,E2 23825.099} C_VEL
LIN {X 0,Y 494.911,Z 1056.139,A -85,B 0,C 180,E1 23823.224,E2 23823.224} C_VEL
LIN {X 0,Y 496.595,Z 1038.217,A -85,B 0,C 180,E1 23821.499,E2 23821.499} C_VEL
LIN {X 0,Y 498.259,Z 1020.06,A -85,B 0,C 180,E1 23820.023,E2 23820.023} C_VEL
LIN {X 0,Y 499.978,Z 999.962,A -85,B 0,C 180,E1 23818.641,E2 23818.641} C_VEL
LIN {X 0,Y 501.73,Z 979.247,A -85,B 0,C 180,E1 23817.449,E2 23817.449} C_VEL
LIN {X 0,Y 503.114,Z 959.268,A -85,B 0,C 180,E1 23816.532,E2 23816.532} C_VEL
LIN {X 0,Y 504.329,Z 938.116,A -85,B 0,C 180,E1 23815.789,E2 23815.789} C_VEL
LIN {X 0,Y 505.204,Z 917.124,A -85,B 0,C 180,E1 23815.254,E2 23815.254} C_VEL
LIN {X 0,Y 508.971,Z 706.029,A -85,B 0,C 180,E1 23811.846,E2 23811.846} C_VEL
LIN {X 0,Y 499.375,Z 690.827,A -85,B 0,C 180,E1 23810.657,E2 23810.657} C_VEL
LIN {X 0,Y 493.788,Z 682.552,A -85,B 0,C 180,E1 23809.943,E2 23809.943} C_VEL
LIN {X 0,Y 491.457,Z 678.843,A -85,B 0,C 180,E1 23809.633,E2 23809.633} C_VEL
LIN {X 0,Y 489.366,Z 675.892,A -85,B 0,C 180,E1 23809.357,E2 23809.357} C_VEL
LIN {X 0,Y 488.895,Z 674.242,A -85,B 0,C 180,E1 23809.174,E2 23809.174} C_VEL
LIN {X 0,Y 488.821,Z 673.825,A -85,B 0,C 180,E1 23808.806,E2 23808.806} C_VEL
LIN {X 0,Y 488.825,Z 673.848,A -85,B 0,C 180,E1 23805.216,E2 23805.216} C_VEL
LIN {X 0,Y 488.821,Z 673.813,A -85,B 0,C 180,E1 23801.665,E2 23801.665} C_VEL
LIN {X 0,Y 488.82,Z 673.818,A -85,B 0,C 180,E1 23798.002,E2 23798.002} C_VEL
LIN {X 0,Y 488.817,Z 673.843,A -85,B 0,C 180,E1 23794.483,E2 23794.483} C_VEL
LIN {X 0,Y 488.828,Z 673.803,A -85,B 0,C 180,E1 23790.891,E2 23790.891} C_VEL
LIN {X 0,Y 488.826,Z 673.837,A -85,B 0,C 180,E1 23787.27,E2 23787.27} C_VEL
LIN {X 0,Y 488.816,Z 673.839,A -85,B 0,C 180,E1 23783.763,E2 23783.763} C_VEL
LIN {X 0,Y 488.832,Z 673.833,A -85,B 0,C 180,E1 23780.223,E2 23780.223} C_VEL
LIN {X 0,Y 488.831,Z 673.838,A -85,B 0,C 180,E1 23776.64,E2 23776.64} C_VEL
LIN {X 0,Y 488.819,Z 673.841,A -85,B 0,C 180,E1 23773.123,E2 23773.123} C_VEL
LIN {X 0,Y 488.83,Z 673.846,A -85,B 0,C 180,E1 23769.537,E2 23769.537} C_VEL
LIN {X 0,Y 488.827,Z 673.831,A -85,B 0,C 180,E1 23765.988,E2 23765.988} C_VEL
LIN {X 0,Y 488.817,Z 673.83,A -85,B 0,C 180,E1 23762.345,E2 23762.345} C_VEL
LIN {X 0,Y 488.821,Z 673.842,A -85,B 0,C 180,E1 23758.828,E2 23758.828} C_VEL
LIN {X 0,Y 488.83,Z 673.842,A -85,B 0,C 180,E1 23755.19,E2 23755.19} C_VEL
LIN {X 0,Y 488.819,Z 673.837,A -85,B 0,C 180,E1 23751.65,E2 23751.65} C_VEL
LIN {X 0,Y 488.815,Z 673.825,A -85,B 0,C 180,E1 23748.077,E2 23748.077} C_VEL
LIN {X 0,Y 488.828,Z 673.841,A -85,B 0,C 180,E1 23744.458,E2 23744.458} C_VEL
LIN {X 0,Y 488.819,Z 673.818,A -85,B 0,C 180,E1 23740.897,E2 23740.897} C_VEL
LIN {X 0,Y 488.815,Z 673.842,A -85,B 0,C 180,E1 23737.385,E2 23737.385} C_VEL
LIN {X 0,Y 488.822,Z 673.837,A -85,B 0,C 180,E1 23733.78,E2 23733.78} C_VEL
LIN {X 0,Y 488.819,Z 673.823,A -85,B 0,C 180,E1 23730.14,E2 23730.14} C_VEL
LIN {X 0,Y 488.815,Z 673.827,A -85,B 0,C 180,E1 23726.567,E2 23726.567} C_VEL
LIN {X 0,Y 488.824,Z 673.833,A -85,B 0,C 180,E1 23723.033,E2 23723.033} C_VEL
LIN {X 0,Y 488.823,Z 673.813,A -85,B 0,C 180,E1 23719.425,E2 23719.425} C_VEL
LIN {X 0,Y 488.855,Z 674.08,A -85,B 0,C 180,E1 23717.751,E2 23717.751} C_VEL
LIN {X 0,Y 490.44,Z 677.761,A -85,B 0,C 180,E1 23717.215,E2 23717.215} C_VEL
LIN {X 0,Y 499.544,Z 697.471,A -85,B 0,C 180,E1 23714.721,E2 23714.721} C_VEL
LIN {X 0,Y 506.962,Z 714.885,A -85,B 0,C 180,E1 23712.721,E2 23712.721} C_VEL
LIN {X 0,Y 505.249,Z 753.113,A -85,B 0,C 180,E1 23710.096,E2 23710.096} C_VEL
LIN {X 0,Y 509.529,Z 781.839,A -85,B 0,C 180,E1 23709.2,E2 23709.2} C_VEL
LIN {X 0,Y 505.867,Z 1013.866,A -85,B 0,C 180,E1 23705.522,E2 23705.522} C_VEL
LIN {X 0,Y 504.933,Z 1065.628,A -85,B 0,C 180,E1 23704.679,E2 23704.679} C_VEL
LIN {X 0,Y 504.021,Z 1086.898,A -85,B 0,C 180,E1 23704.139,E2 23704.139} C_VEL
LIN {X 0,Y 502.809,Z 1109.223,A -85,B 0,C 180,E1 23703.365,E2 23703.365} C_VEL
LIN {X 0,Y 501.54,Z 1130.254,A -85,B 0,C 180,E1 23702.429,E2 23702.429} C_VEL
LIN {X 0,Y 500.046,Z 1149.007,A -85,B 0,C 180,E1 23701.373,E2 23701.373} C_VEL
LIN {X 0,Y 498.309,Z 1169.503,A -85,B 0,C 180,E1 23699.974,E2 23699.974} C_VEL
LIN {X 0,Y 496.643,Z 1187.76,A -85,B 0,C 180,E1 23698.498,E2 23698.498} C_VEL
LIN {X 0,Y 494.931,Z 1205.873,A -85,B 0,C 180,E1 23696.757,E2 23696.757} C_VEL
LIN {X 0,Y 493.328,Z 1222.674,A -85,B 0,C 180,E1 23694.869,E2 23694.869} C_VEL
LIN {X 0,Y 491.924,Z 1238.18,A -85,B 0,C 180,E1 23692.843,E2 23692.843} C_VEL
LIN {X 0,Y 490.706,Z 1252.634,A -85,B 0,C 180,E1 23690.64,E2 23690.64} C_VEL
LIN {X 0,Y 489.722,Z 1265.455,A -85,B 0,C 180,E1 23688.325,E2 23688.325} C_VEL
LIN {X 0,Y 488.979,Z 1276.813,A -85,B 0,C 180,E1 23685.902,E2 23685.902} C_VEL
LIN {X 0,Y 488.493,Z 1286.26,A -85,B 0,C 180,E1 23683.493,E2 23683.493} C_VEL
LIN {X 0,Y 488.183,Z 1293.882,A -85,B 0,C 180,E1 23681.1,E2 23681.1} C_VEL
LIN {X 0,Y 488.006,Z 1300.146,A -85,B 0,C 180,E1 23678.602,E2 23678.602} C_VEL
LIN {X 0,Y 487.93,Z 1304.636,A -85,B 0,C 180,E1 23676.235,E2 23676.235} C_VEL
LIN {X 0,Y 487.901,Z 1307.674,A -85,B 0,C 180,E1 23673.76,E2 23673.76} C_VEL
LIN {X 0,Y 487.908,Z 1309.282,A -85,B 0,C 180,E1 23671.174,E2 23671.174} C_VEL
LIN {X 0,Y 487.908,Z 1309.281,A -85,B 0,C 180,E1 23668.826,E2 23668.826} C_VEL
LIN {X 0,Y 487.901,Z 1307.672,A -85,B 0,C 180,E1 23666.24,E2 23666.24} C_VEL
LIN {X 0,Y 487.93,Z 1304.633,A -85,B 0,C 180,E1 23663.765,E2 23663.765} C_VEL
LIN {X 0,Y 488.006,Z 1300.145,A -85,B 0,C 180,E1 23661.398,E2 23661.398} C_VEL
LIN {X 0,Y 488.195,Z 1293.529,A -85,B 0,C 180,E1 23658.781,E2 23658.781} C_VEL
LIN {X 0,Y 488.516,Z 1285.85,A -85,B 0,C 180,E1 23656.387,E2 23656.387} C_VEL
LIN {X 0,Y 489.024,Z 1276.126,A -85,B 0,C 180,E1 23653.937,E2 23653.937} C_VEL
LIN {X 0,Y 489.766,Z 1264.821,A -85,B 0,C 180,E1 23651.553,E2 23651.553} C_VEL
LIN {X 0,Y 490.706,Z 1252.634,A -85,B 0,C 180,E1 23649.36,E2 23649.36} C_VEL
LIN {X 0,Y 491.924,Z 1238.18,A -85,B 0,C 180,E1 23647.157,E2 23647.157} C_VEL
LIN {X 0,Y 493.328,Z 1222.675,A -85,B 0,C 180,E1 23645.131,E2 23645.131} C_VEL
LIN {X 0,Y 494.946,Z 1205.705,A -85,B 0,C 180,E1 23643.226,E2 23643.226} C_VEL
LIN {X 0,Y 496.645,Z 1187.762,A -85,B 0,C 180,E1 23641.503,E2 23641.503} C_VEL
LIN {X 0,Y 498.311,Z 1169.509,A -85,B 0,C 180,E1 23640.026,E2 23640.026} C_VEL
LIN {X 0,Y 500.046,Z 1149.01,A -85,B 0,C 180,E1 23638.627,E2 23638.627} C_VEL
LIN {X 0,Y 501.539,Z 1130.254,A -85,B 0,C 180,E1 23637.571,E2 23637.571} C_VEL
LIN {X 0,Y 502.811,Z 1109.228,A -85,B 0,C 180,E1 23636.635,E2 23636.635} C_VEL
LIN {X 0,Y 504.053,Z 1086.28,A -85,B 0,C 180,E1 23635.843,E2 23635.843} C_VEL
LIN {X 0,Y 504.959,Z 1064.936,A -85,B 0,C 180,E1 23635.306,E2 23635.306} C_VEL
LIN {X 0,Y 506.332,Z 983.06,A -85,B 0,C 180,E1 23633.995,E2 23633.995} C_VEL
LIN {X 0,Y 509.491,Z 780.348,A -85,B 0,C 180,E1 23630.77,E2 23630.77} C_VEL
LIN {X 0,Y 505.191,Z 752.122,A -85,B 0,C 180,E1 23629.857,E2 23629.857} C_VEL
LIN {X 0,Y 506.956,Z 714.35,A -85,B 0,C 180,E1 23627.238,E2 23627.238} C_VEL
LIN {X 0,Y 495.765,Z 689.084,A -85,B 0,C 180,E1 23624.251,E2 23624.251} C_VEL
LIN {X 0,Y 489.889,Z 676.888,A -85,B 0,C 180,E1 23622.657,E2 23622.657} C_VEL
LIN {X 0,Y 488.844,Z 674.01,A -85,B 0,C 180,E1 23622.235,E2 23622.235} C_VEL
LIN {X 0,Y 488.815,Z 673.838,A -85,B 0,C 180,E1 23618.749,E2 23618.749} C_VEL
LIN {X 0,Y 488.822,Z 673.841,A -85,B 0,C 180,E1 23615.227,E2 23615.227} C_VEL
LIN {X 0,Y 488.824,Z 673.844,A -85,B 0,C 180,E1 23611.576,E2 23611.576} C_VEL
LIN {X 0,Y 488.817,Z 673.842,A -85,B 0,C 180,E1 23608.064,E2 23608.064} C_VEL
LIN {X 0,Y 488.82,Z 673.824,A -85,B 0,C 180,E1 23604.467,E2 23604.467} C_VEL
LIN {X 0,Y 488.824,Z 673.84,A -85,B 0,C 180,E1 23600.815,E2 23600.815} C_VEL
